C03642=1046.067,28.309,420.104,170.138,34.903,156.571
C03643=1046.061,28.059,420.121,170.136,34.901,156.571
C03644=1046.054,27.810,420.136,170.135,34.900,156.571
C03645=1046.047,27.560,420.153,170.133,34.899,156.571
C03646=1046.041,27.311,420.169,170.131,34.897,156.570
C03647=1046.035,27.062,420.185,170.130,34.895,156.570
C03648=1046.029,26.813,420.201,170.128,34.894,156.570
C03649=1046.022,26.564,420.217,170.126,34.893,156.570
C03650=1046.016,26.314,420.233,170.124,34.891,156.569
C03651=1046.010,26.064,420.250,170.123,34.889,156.569
C03652=1046.003,25.815,420.265,170.121,34.888,156.569
C03653=1045.997,25.566,420.281,170.119,34.887,156.569
C03654=1045.991,25.316,420.296,170.116,34.885,156.568
C03655=1045.985,25.067,420.313,170.115,34.883,156.568
C03656=1045.978,24.818,420.328,170.113,34.882,156.568
C03657=1045.971,24.568,420.345,170.111,34.881,156.568
C03658=1045.965,24.318,420.361,170.109,34.879,156.567
C03659=1045.959,24.069,420.377,170.108,34.878,156.567
C03660=1045.953,23.820,420.393,170.106,34.876,156.567
C03661=1045.946,23.570,420.408,170.104,34.875,156.567
C03662=1045.940,23.321,420.424,170.102,34.873,156.566
C03663=1045.934,23.072,420.440,170.101,34.872,156.566
C03664=1045.928,22.823,420.456,170.099,34.870,156.566
C03665=1045.921,22.572,420.473,170.097,34.869,156.566
C03666=1045.915,22.323,420.488,170.096,34.868,156.565
C03667=1045.909,22.073,420.504,170.094,34.866,156.565
C03668=1045.902,21.824,420.520,170.091,34.864,156.565
C03669=1045.896,21.575,420.536,170.089,34.863,156.565
C03670=1045.890,21.325,420.551,170.088,34.862,156.564
C03671=1045.884,21.076,420.567,170.086,34.860,156.564
C03672=1045.877,20.827,420.583,170.084,34.858,156.564
C03673=1045.871,20.578,420.599,170.082,34.857,156.564
C03674=1045.866,20.328,420.615,170.081,34.856,156.564
C03675=1045.859,20.079,420.630,170.079,34.854,156.563
C03676=1045.853,19.829,420.647,170.077,34.852,156.563
C03677=1045.846,19.579,420.662,170.075,34.851,156.563
C03678=1045.839,19.330,420.678,170.074,34.850,156.563
C03679=1045.833,19.081,420.694,170.072,34.848,156.562
C03680=1045.827,18.831,420.709,170.070,34.847,156.562
C03681=1045.821,18.582,420.725,170.068,34.846,156.562
C03682=1045.814,18.333,420.741,170.066,34.844,156.562
C03683=1045.808,18.083,420.756,170.064,34.842,156.561
C03684=1045.802,17.834,420.772,170.062,34.841,156.561
C03685=1045.795,17.585,420.788,170.060,34.840,156.561
C03686=1045.790,17.335,420.803,170.058,34.838,156.561
C03687=1045.783,17.086,420.819,170.057,34.837,156.561
C03688=1045.777,16.836,420.834,170.055,34.835,156.560
C03689=1045.771,16.586,420.850,170.053,34.834,156.560
C03690=1045.764,16.337,420.866,170.051,34.832,156.560
C03691=1045.758,16.087,420.881,170.050,34.831,156.560
C03692=1045.752,15.838,420.897,170.048,34.830,156.559
C03693=1045.745,15.589,420.912,170.046,34.828,156.559
C03694=1045.739,15.339,420.928,170.044,34.827,156.559
C03695=1045.733,15.090,420.943,170.043,34.825,156.559
C03696=1045.727,14.840,420.959,170.040,34.824,156.558
C03697=1045.721,14.591,420.974,170.038,34.823,156.558
C03698=1045.714,14.342,420.990,170.036,34.821,156.558
C03699=1045.708,14.092,421.005,170.035,34.820,156.558
C03700=1045.702,13.843,421.021,170.033,34.819,156.558
C03701=1045.695,13.593,421.036,170.031,34.817,156.557
C03702=1045.688,13.308,421.054,170.029,34.815,156.557
C03703=1045.680,13.023,421.071,170.027,34.814,156.557
C03704=1045.673,12.737,421.089,170.025,34.813,156.557
C03705=1045.666,12.453,421.106,170.023,34.811,156.556
C03706=1045.659,12.203,421.121,170.021,34.809,156.556
C03707=1045.653,11.954,421.138,170.019,34.808,156.556
C03708=1045.647,11.704,421.152,170.017,34.807,156.556
C03709=1045.640,11.455,421.167,170.015,34.805,156.555
C03710=1045.634,11.206,421.183,170.014,34.804,156.555
C03711=1045.627,10.956,421.198,170.011,34.803,156.555
C03712=1045.621,10.707,421.214,170.009,34.801,156.555
C03713=1045.614,10.457,421.229,170.007,34.800,156.555
C03714=1045.609,10.207,421.244,170.005,34.798,156.554
C03715=1045.602,9.958,421.260,170.004,34.797,156.554
C03716=1045.596,9.709,421.275,170.002,34.796,156.554
C03717=1045.589,9.459,421.290,170.000,34.795,156.554
C03718=1045.583,9.210,421.305,169.998,34.793,156.554
C03719=1045.576,8.960,421.320,169.996,34.792,156.553
C03720=1045.570,8.711,421.335,169.995,34.791,156.553
C03721=1045.563,8.462,421.351,169.993,34.789,156.553
C03722=1045.557,8.212,421.367,169.991,34.788,156.553
C03723=1045.551,7.962,421.381,169.989,34.786,156.552
C03724=1045.545,7.712,421.396,169.987,34.785,156.552
C03725=1045.538,7.463,421.412,169.986,34.783,156.552
C03726=1045.532,7.214,421.427,169.984,34.782,156.552
C03727=1045.526,6.965,421.442,169.981,34.780,156.552
C03728=1045.519,6.715,421.457,169.979,34.779,156.551
C03729=1045.513,6.466,421.472,169.977,34.778,156.551
C03730=1045.506,6.216,421.487,169.975,34.776,156.551
C03731=1045.501,5.966,421.503,169.974,34.775,156.551
C03732=1045.494,5.717,421.518,169.972,34.774,156.550
C03733=1045.488,5.468,421.533,169.970,34.772,156.550
C03734=1045.482,5.219,421.548,169.968,34.771,156.550
C03735=1045.476,4.969,421.563,169.966,34.770,156.550
C03736=1045.469,4.719,421.578,169.965,34.768,156.550
C03737=1045.463,4.470,421.593,169.963,34.767,156.549
C03738=1045.456,4.220,421.608,169.961,34.766,156.549
C03739=1045.450,3.971,421.623,169.959,34.764,156.549
C03740=1045.443,3.721,421.638,169.957,34.763,156.549
C03741=1045.437,3.472,421.653,169.955,34.762,156.549
C03742=1045.432,3.222,421.668,169.954,34.760,156.548
C03743=1045.425,2.973,421.683,169.952,34.759,156.548
C03744=1045.419,2.723,421.698,169.949,34.758,156.548
C03745=1045.413,2.473,421.713,169.947,34.756,156.548
C03746=1045.407,2.225,421.729,169.945,34.755,156.548
C03747=1045.400,1.975,421.743,169.943,34.754,156.547
C03748=1045.394,1.726,421.758,169.942,34.752,156.547
C03749=1045.387,1.476,421.773,169.940,34.751,156.547
C03750=1045.381,1.226,421.788,169.938,34.750,156.547
C03751=1045.375,0.977,421.803,169.936,34.748,156.546
C03752=1045.369,0.728,421.818,169.934,34.746,156.546
C03753=1045.363,0.478,421.833,169.932,34.745,156.546
C03754=1045.356,0.229,421.848,169.931,34.744,156.546
C03755=1045.350,-0.020,421.862,169.929,34.742,156.546
C03756=1045.344,-0.270,421.877,169.927,34.741,156.545
C03757=1045.338,-0.520,421.892,169.925,34.740,156.545
C03758=1045.332,-0.770,421.908,169.923,34.738,156.545
C03759=1045.326,-1.019,421.922,169.921,34.737,156.545
C03760=1045.320,-1.268,421.937,169.920,34.736,156.545
C03761=1045.313,-1.518,421.952,169.917,34.734,156.544
C03762=1045.307,-1.768,421.967,169.915,34.733,156.544
C03763=1045.301,-2.017,421.982,169.913,34.732,156.544
C03764=1045.295,-2.266,421.997,169.911,34.730,156.544
C03765=1045.288,-2.516,422.012,169.909,34.729,156.543
C03766=1045.281,-2.799,422.029,169.907,34.727,156.543
C03767=1045.274,-3.082,422.045,169.905,34.725,156.543
C03768=1045.267,-3.365,422.063,169.903,34.724,156.543
C03769=1045.260,-3.649,422.079,169.901,34.723,156.543
C03770=1045.254,-3.898,422.093,169.899,34.721,156.542
C03771=1045.247,-4.147,422.108,169.897,34.720,156.542
C03772=1045.241,-4.397,422.122,169.895,34.719,156.542
C03773=1045.235,-4.647,422.137,169.894,34.717,156.542
C03774=1045.228,-4.896,422.151,169.892,34.717,156.542
C03775=1045.222,-5.145,422.166,169.890,34.715,156.541
C03776=1045.216,-5.395,422.181,169.888,34.714,156.541
C03777=1045.209,-5.645,422.196,169.886,34.713,156.541
C03778=1045.203,-5.894,422.209,169.884,34.711,156.541
C03779=1045.197,-6.144,422.224,169.881,34.710,156.541
C03780=1045.190,-6.393,422.239,169.879,34.709,156.540
C03781=1045.184,-6.642,422.253,169.877,34.708,156.540
C03782=1045.177,-6.892,422.268,169.876,34.706,156.540
C03783=1045.171,-7.142,422.282,169.874,34.705,156.540
C03784=1045.165,-7.392,422.297,169.872,34.704,156.540
C03785=1045.158,-7.640,422.311,169.870,34.702,156.539
C03786=1045.152,-7.890,422.326,169.868,34.701,156.539
C03787=1045.146,-8.140,422.340,169.866,34.700,156.539
C03788=1045.139,-8.389,422.354,169.864,34.699,156.539
C03789=1045.133,-8.638,422.369,169.862,34.698,156.539
C03790=1045.127,-8.888,422.384,169.860,34.696,156.539
C03791=1045.121,-9.138,422.398,169.858,34.695,156.538
C03792=1045.114,-9.387,422.413,169.857,34.694,156.538
C03793=1045.108,-9.637,422.427,169.855,34.692,156.538
C03794=1045.102,-9.886,422.441,169.853,34.692,156.538
C03795=1045.095,-10.136,422.456,169.851,34.690,156.538
C03796=1045.089,-10.385,422.470,169.849,34.689,156.537
C03797=1045.083,-10.635,422.484,169.847,34.687,156.537
C03798=1045.076,-10.884,422.499,169.845,34.686,156.537
C03799=1045.070,-11.133,422.513,169.842,34.685,156.537
C03800=1045.064,-11.383,422.528,169.840,34.684,156.537
C03801=1045.058,-11.633,422.543,169.838,34.683,156.536
C03802=1045.052,-11.882,422.556,169.837,34.681,156.536
C03803=1045.045,-12.132,422.571,169.835,34.680,156.536
C03804=1045.039,-12.381,422.585,169.833,34.679,156.536
C03805=1045.033,-12.631,422.599,169.831,34.677,156.536
C03806=1045.027,-12.880,422.614,169.829,34.677,156.536
C03807=1045.021,-13.130,422.628,169.827,34.675,156.535
C03808=1045.014,-13.379,422.642,169.825,34.674,156.535
C03809=1045.008,-13.628,422.657,169.823,34.672,156.535
C03810=1045.002,-13.879,422.671,169.821,34.671,156.535
C03811=1044.995,-14.127,422.685,169.819,34.670,156.535
C03812=1044.989,-14.378,422.699,169.817,34.669,156.534
C03813=1044.983,-14.627,422.714,169.816,34.668,156.534
C03814=1044.977,-14.877,422.727,169.814,34.666,156.534
C03815=1044.971,-15.125,422.742,169.812,34.665,156.534
C03816=1044.964,-15.375,422.756,169.810,34.664,156.534
C03817=1044.958,-15.625,422.771,169.808,34.663,156.534
C03818=1044.951,-15.874,422.784,169.806,34.662,156.533
C03819=1044.945,-16.124,422.799,169.804,34.660,156.533
C03820=1044.939,-16.373,422.812,169.801,34.659,156.533
C03821=1044.933,-16.624,422.826,169.799,34.658,156.533
C03822=1044.926,-16.872,422.840,169.797,34.657,156.533
C03823=1044.919,-17.122,422.854,169.795,34.656,156.533
C03824=1044.913,-17.372,422.869,169.793,34.655,156.532
C03825=1044.907,-17.621,422.882,169.791,34.653,156.532
C03826=1044.900,-17.871,422.897,169.789,34.653,156.532
C03827=1044.894,-18.120,422.910,169.787,34.651,156.532
C03828=1044.888,-18.370,422.925,169.785,34.650,156.532
C03829=1044.882,-18.619,422.939,169.783,34.648,156.531
C03830=1044.874,-18.901,422.954,169.781,34.648,156.531
C03831=1044.867,-19.183,422.970,169.779,34.646,156.531
C03832=1044.860,-19.464,422.986,169.777,34.645,156.531
C03833=1044.853,-19.745,423.002,169.775,34.644,156.531
C03834=1044.847,-19.996,423.016,169.773,34.642,156.530
C03835=1044.841,-20.245,423.029,169.771,34.642,156.530
C03836=1044.834,-20.495,423.043,169.769,34.640,156.530
C03837=1044.828,-20.744,423.057,169.767,34.639,156.530
C03838=1044.821,-20.994,423.071,169.765,34.638,156.530
C03839=1044.816,-21.243,423.085,169.763,34.637,156.530
C03840=1044.809,-21.493,423.099,169.761,34.635,156.529
C03841=1044.803,-21.742,423.112,169.759,34.635,156.529
C03842=1044.796,-21.992,423.127,169.757,34.633,156.529
C03843=1044.790,-22.242,423.140,169.755,34.632,156.529
C03844=1044.784,-22.491,423.154,169.752,34.631,156.529
C03845=1044.778,-22.741,423.168,169.750,34.630,156.529
C03846=1044.771,-22.990,423.181,169.748,34.628,156.528
C03847=1044.765,-23.240,423.196,169.746,34.628,156.528
C03848=1044.759,-23.489,423.210,169.744,34.626,156.528
C03849=1044.752,-23.739,423.223,169.742,34.625,156.528
C03850=1044.747,-23.988,423.237,169.740,34.624,156.528
C03851=1044.740,-24.238,423.250,169.738,34.623,156.528
C03852=1044.734,-24.488,423.265,169.736,34.621,156.527
C03853=1044.728,-24.736,423.279,169.734,34.621,156.527
C03854=1044.721,-24.986,423.292,169.732,34.619,156.527
C03855=1044.715,-25.236,423.306,169.730,34.618,156.527
C03856=1044.709,-25.485,423.319,169.728,34.617,156.527
C03857=1044.702,-25.735,423.333,169.726,34.616,156.527
C03858=1044.697,-25.985,423.347,169.724,34.615,156.527
C03859=1044.691,-26.234,423.360,169.722,34.614,156.526
C03860=1044.684,-26.483,423.374,169.720,34.612,156.526
C03861=1044.678,-26.733,423.388,169.718,34.611,156.526
C03862=1044.672,-26.982,423.402,169.716,34.610,156.526
C03863=1044.665,-27.232,423.415,169.714,34.609,156.526
C03864=1044.659,-27.481,423.428,169.712,34.608,156.526
C03865=1044.653,-27.732,423.443,169.710,34.607,156.525
C03866=1044.647,-27.981,423.456,169.708,34.606,156.525
C03867=1044.640,-28.230,423.469,169.706,34.605,156.525
C03868=1044.634,-28.480,423.483,169.704,34.604,156.525
C03869=1044.627,-28.729,423.496,169.702,34.603,156.525
C03870=1044.621,-28.979,423.510,169.700,34.602,156.525
C03871=1044.614,-29.229,423.523,169.697,34.601,156.525
C03872=1044.608,-29.478,423.536,169.695,34.600,156.524
C03873=1044.601,-29.728,423.550,169.693,34.598,156.524
C03874=1044.596,-29.978,423.564,169.691,34.598,156.524
C03875=1044.590,-30.227,423.577,169.689,34.596,156.524
C03876=1044.583,-30.477,423.591,169.687,34.596,156.524
C03877=1044.577,-30.726,423.604,169.685,34.594,156.524
C03878=1044.570,-30.975,423.617,169.683,34.594,156.524
C03879=1044.564,-31.225,423.631,169.681,34.593,156.523
C03880=1044.557,-31.475,423.644,169.679,34.591,156.523
C03881=1044.551,-31.724,423.657,169.677,34.591,156.523
C03882=1044.545,-31.974,423.670,169.675,34.589,156.523
C03883=1044.539,-32.224,423.684,169.673,34.589,156.523
C03884=1044.533,-32.473,423.698,169.671,34.587,156.523
C03885=1044.527,-32.722,423.711,169.669,34.587,156.523
C03886=1044.520,-32.972,423.724,169.667,34.585,156.522
C03887=1044.514,-33.222,423.738,169.665,34.584,156.522
C03888=1044.507,-33.471,423.751,169.663,34.583,156.522
C03889=1044.501,-33.721,423.765,169.660,34.582,156.522
C03890=1044.495,-33.971,423.777,169.658,34.581,156.522
C03891=1044.488,-34.220,423.790,169.656,34.580,156.522
C03892=1044.482,-34.469,423.804,169.654,34.579,156.522
C03893=1044.475,-34.719,423.817,169.652,34.578,156.521
C03894=1044.468,-35.047,423.834,169.650,34.577,156.521
C03895=1044.460,-35.375,423.852,169.647,34.575,156.521
C03896=1044.451,-35.704,423.869,169.644,34.574,156.521
C03897=1044.443,-36.032,423.887,169.642,34.572,156.521
C03898=1044.437,-36.258,423.898,169.640,34.572,156.521
C03899=1044.432,-36.484,423.911,169.638,34.571,156.520
C03900=1044.426,-36.710,423.923,169.636,34.570,156.520
C03901=1044.421,-36.935,423.934,169.634,34.569,156.520
C03902=1044.415,-37.161,423.947,169.632,34.568,156.520
C03903=1044.410,-37.387,423.959,169.630,34.567,156.520
C03904=1044.404,-37.613,423.971,169.628,34.566,156.520
C03905=1044.398,-37.839,423.982,169.626,34.565,156.520
C03906=1044.392,-38.089,423.996,169.624,34.564,156.520
C03907=1044.385,-38.338,424.009,169.622,34.563,156.519
C03908=1044.379,-38.588,424.021,169.619,34.562,156.519
C03909=1044.373,-38.837,424.035,169.617,34.561,156.519
C03910=1044.367,-39.087,424.048,169.615,34.560,156.519
C03911=1044.361,-39.337,424.061,169.613,34.560,156.519
C03912=1044.354,-39.586,424.074,169.611,34.558,156.519
C03913=1044.348,-39.836,424.087,169.609,34.557,156.519
C03914=1044.341,-40.085,424.099,169.607,34.557,156.519
C03915=1044.335,-40.335,424.113,169.605,34.556,156.518
C03916=1044.329,-40.584,424.125,169.603,34.555,156.518
C03917=1044.322,-40.834,424.139,169.601,34.554,156.518
C03918=1044.317,-41.084,424.151,169.599,34.553,156.518
C03919=1044.310,-41.333,424.164,169.596,34.552,156.518
C03920=1044.303,-41.583,424.177,169.594,34.551,156.518
C03921=1044.298,-41.832,424.190,169.592,34.550,156.518
C03922=1044.291,-42.082,424.203,169.590,34.549,156.518
C03923=1044.285,-42.332,424.216,169.588,34.548,156.517
C03924=1044.279,-42.582,424.229,169.586,34.547,156.517
C03925=1044.272,-42.831,424.241,169.584,34.547,156.517
C03926=1044.266,-43.080,424.255,169.582,34.546,156.517
C03927=1044.260,-43.330,424.267,169.580,34.545,156.517
C03928=1044.254,-43.579,424.280,169.578,34.544,156.517
C03929=1044.247,-43.829,424.292,169.575,34.543,156.517
C03930=1044.241,-44.078,424.306,169.573,34.542,156.517
C03931=1044.234,-44.329,424.319,169.571,34.541,156.517
C03932=1044.228,-44.578,424.332,169.569,34.540,156.516
C03933=1044.222,-44.828,424.344,169.567,34.539,156.516
C03934=1044.215,-45.077,424.357,169.565,34.539,156.516
C03935=1044.209,-45.327,424.370,169.563,34.537,156.516
C03936=1044.203,-45.577,424.382,169.561,34.537,156.516
C03937=1044.197,-45.826,424.395,169.559,34.536,156.516
C03938=1044.190,-46.076,424.407,169.556,34.535,156.516
C03939=1044.184,-46.325,424.421,169.554,34.534,156.516
C03940=1044.178,-46.575,424.433,169.552,34.533,156.516
C03941=1044.172,-46.825,424.446,169.550,34.532,156.515
C03942=1044.166,-47.074,424.459,169.548,34.531,156.515
C03943=1044.160,-47.323,424.471,169.546,34.531,156.515
C03944=1044.153,-47.573,424.484,169.544,34.529,156.515
C03945=1044.147,-47.823,424.497,169.542,34.529,156.515
C03946=1044.142,-48.073,424.509,169.540,34.528,156.515
C03947=1044.135,-48.321,424.522,169.537,34.527,156.515
C03948=1044.129,-48.571,424.535,169.534,34.526,156.515
C03949=1044.123,-48.821,424.547,169.532,34.525,156.515
C03950=1044.117,-49.070,424.560,169.530,34.524,156.514
C03951=1044.110,-49.320,424.572,169.528,34.523,156.514
C03952=1044.104,-49.570,424.585,169.526,34.523,156.514
C03953=1044.098,-49.819,424.598,169.524,34.521,156.514
C03954=1044.092,-50.069,424.611,169.522,34.521,156.514
C03955=1044.085,-50.319,424.623,169.519,34.520,156.514
C03956=1044.079,-50.569,424.635,169.517,34.519,156.514
C03957=1044.073,-50.818,424.647,169.515,34.518,156.514
C03958=1044.065,-51.100,424.662,169.513,34.518,156.514
C03959=1044.058,-51.381,424.676,169.510,34.517,156.514
C03960=1044.052,-51.662,424.689,169.508,34.516,156.513
C03961=1044.043,-51.943,424.703,169.505,34.515,156.513
C03962=1044.038,-52.193,424.716,169.503,34.514,156.513
C03963=1044.031,-52.443,424.728,169.501,34.514,156.513
C03964=1044.025,-52.692,424.741,169.499,34.513,156.513
C03965=1044.018,-52.942,424.753,169.497,34.512,156.513
C03966=1044.011,-53.191,424.765,169.494,34.511,156.513
C03967=1044.005,-53.441,424.778,169.492,34.511,156.513
C03968=1043.999,-53.691,424.790,169.490,34.510,156.513
C03969=1043.993,-53.941,424.802,169.488,34.509,156.513
C03970=1043.986,-54.190,424.814,169.486,34.508,156.513
C03971=1043.980,-54.440,424.826,169.483,34.508,156.513
C03972=1043.974,-54.690,424.839,169.481,34.507,156.512
C03973=1043.967,-54.939,424.851,169.479,34.506,156.512
C03974=1043.960,-55.188,424.863,169.477,34.505,156.512
C03975=1043.954,-55.438,424.876,169.475,34.505,156.512
C03976=1043.948,-55.688,424.888,169.473,34.504,156.512
C03977=1043.942,-55.937,424.900,169.470,34.503,156.512
C03978=1043.935,-56.187,424.912,169.468,34.502,156.512
C03979=1043.928,-56.437,424.924,169.466,34.502,156.512
C03980=1043.923,-56.686,424.936,169.464,34.501,156.512
C03981=1043.916,-56.935,424.948,169.462,34.501,156.512
C03982=1043.910,-57.185,424.960,169.459,34.500,156.512
C03983=1043.904,-57.435,424.973,169.457,34.499,156.512
C03984=1043.897,-57.684,424.985,169.455,34.499,156.512
C03985=1043.891,-57.934,424.997,169.453,34.498,156.511
C03986=1043.885,-58.184,425.009,169.451,34.497,156.511
C03987=1043.878,-58.433,425.021,169.448,34.496,156.511
C03988=1043.872,-58.683,425.034,169.446,34.495,156.511
C03989=1043.866,-58.933,425.045,169.444,34.495,156.511
C03990=1043.860,-59.182,425.057,169.442,34.494,156.511
C03991=1043.854,-59.432,425.069,169.440,34.493,156.511
C03992=1043.847,-59.682,425.081,169.437,34.493,156.511
C03993=1043.840,-59.931,425.093,169.435,34.492,156.511
C03994=1043.835,-60.181,425.106,169.433,34.492,156.511
C03995=1043.828,-60.431,425.118,169.431,34.491,156.511
C03996=1043.822,-60.680,425.129,169.429,34.490,156.511
C03997=1043.816,-60.930,425.142,169.426,34.489,156.511
C03998=1043.809,-61.179,425.154,169.424,34.489,156.510
C03999=1043.803,-61.429,425.165,169.422,34.488,156.510
C04000=1043.797,-61.679,425.178,169.420,34.487,156.510
C04001=1043.791,-61.928,425.189,169.418,34.487,156.510
C04002=1043.784,-62.178,425.201,169.415,34.486,156.510
C04003=1043.778,-62.428,425.214,169.413,34.485,156.510
C04004=1043.772,-62.677,425.226,169.411,34.485,156.510
C04005=1043.765,-62.927,425.237,169.409,34.484,156.510
C04006=1043.760,-63.177,425.249,169.406,34.483,156.510
C04007=1043.754,-63.426,425.261,169.404,34.482,156.510
C04008=1043.747,-63.676,425.273,169.402,34.482,156.510
C04009=1043.740,-63.925,425.285,169.400,34.482,156.510
C04010=1043.735,-64.175,425.296,169.398,34.481,156.510
C04011=1043.729,-64.425,425.308,169.395,34.480,156.510
C04012=1043.722,-64.674,425.320,169.393,34.479,156.509
C04013=1043.716,-64.924,425.333,169.391,34.479,156.509
C04014=1043.710,-65.174,425.344,169.389,34.478,156.509
C04015=1043.704,-65.423,425.356,169.386,34.478,156.509
C04016=1043.698,-65.673,425.368,169.384,34.477,156.509
C04017=1043.691,-65.923,425.380,169.382,34.476,156.509
C04018=1043.685,-66.172,425.391,169.380,34.475,156.509
C04019=1043.679,-66.422,425.403,169.378,34.475,156.509
C04020=1043.673,-66.672,425.416,169.375,34.474,156.509
C04021=1043.667,-66.921,425.426,169.373,34.474,156.509
C04022=1043.659,-67.204,425.441,169.371,34.473,156.509
C04023=1043.653,-67.486,425.454,169.368,34.472,156.509
C04024=1043.646,-67.769,425.467,169.366,34.471,156.509
C04025=1043.639,-68.051,425.480,169.363,34.471,156.509
C04026=1043.633,-68.301,425.492,169.361,34.470,156.509
C04027=1043.627,-68.550,425.503,169.359,34.469,156.508
C04028=1043.621,-68.800,425.516,169.356,34.469,156.509
C04029=1043.614,-69.050,425.527,169.354,34.468,156.508
C04030=1043.608,-69.299,425.539,169.352,34.467,156.508
C04031=1043.603,-69.550,425.550,169.350,34.467,156.508
C04032=1043.596,-69.799,425.562,169.347,34.467,156.508
C04033=1043.590,-70.049,425.573,169.345,34.466,156.508
C04034=1043.584,-70.298,425.585,169.343,34.465,156.508
C04035=1043.578,-70.548,425.597,169.341,34.464,156.508
C04036=1043.572,-70.798,425.609,169.338,34.463,156.508
C04037=1043.565,-71.047,425.621,169.336,34.463,156.508
C04038=1043.560,-71.297,425.631,169.334,34.463,156.508
C04039=1043.553,-71.546,425.643,169.332,34.462,156.508
C04040=1043.548,-71.796,425.655,169.329,34.461,156.508
C04041=1043.541,-72.046,425.667,169.327,34.461,156.508
C04042=1043.535,-72.296,425.678,169.325,34.460,156.508
C04043=1043.529,-72.545,425.690,169.323,34.459,156.508
C04044=1043.523,-72.795,425.701,169.320,34.459,156.508
C04045=1043.517,-73.044,425.713,169.318,34.459,156.508
C04046=1043.511,-73.294,425.724,169.316,34.458,156.507
C04047=1043.505,-73.543,425.736,169.314,34.457,156.507
C04048=1043.499,-73.794,425.748,169.311,34.456,156.507
C04049=1043.493,-74.044,425.759,169.309,34.456,156.507
C04050=1043.487,-74.293,425.771,169.307,34.455,156.507
C04051=1043.481,-74.543,425.782,169.305,34.455,156.507
C04052=1043.474,-74.792,425.793,169.302,34.455,156.507
C04053=1043.468,-75.042,425.805,169.300,34.454,156.507
C04054=1043.462,-75.292,425.816,169.298,34.454,156.507
C04055=1043.456,-75.541,425.827,169.295,34.453,156.507
C04056=1043.449,-75.791,425.839,169.293,34.453,156.507
C04057=1043.444,-76.041,425.850,169.291,34.452,156.507
C04058=1043.436,-76.290,425.861,169.289,34.452,156.507
C04059=1043.431,-76.540,425.872,169.286,34.451,156.507
C04060=1043.424,-76.790,425.883,169.284,34.451,156.507
C04061=1043.418,-77.039,425.895,169.282,34.450,156.507
C04062=1043.412,-77.289,425.906,169.279,34.450,156.507
C04063=1043.406,-77.538,425.917,169.277,34.449,156.507
C04064=1043.399,-77.788,425.929,169.275,34.449,156.507
C04065=1043.394,-78.037,425.940,169.272,34.448,156.507
C04066=1043.387,-78.288,425.951,169.270,34.448,156.507
C04067=1043.382,-78.537,425.962,169.268,34.448,156.507
C04068=1043.375,-78.787,425.974,169.266,34.447,156.507
C04069=1043.369,-79.036,425.985,169.263,34.447,156.507
C04070=1043.363,-79.286,425.996,169.261,34.446,156.507
C04071=1043.357,-79.536,426.007,169.259,34.446,156.507
C04072=1043.351,-79.786,426.018,169.256,34.445,156.507
C04073=1043.345,-80.035,426.030,169.254,34.445,156.507
C04074=1043.338,-80.285,426.040,169.252,34.445,156.507
C04075=1043.331,-80.535,426.051,169.249,34.444,156.507
C04076=1043.326,-80.784,426.062,169.247,34.444,156.507
C04077=1043.319,-81.034,426.073,169.245,34.444,156.507
C04078=1043.313,-81.284,426.084,169.242,34.443,156.506
C04079=1043.306,-81.534,426.095,169.240,34.443,156.507
C04080=1043.301,-81.783,426.106,169.238,34.443,156.507
C04081=1043.293,-82.033,426.117,169.235,34.442,156.506
C04082=1043.288,-82.282,426.128,169.233,34.442,156.507
C04083=1043.282,-82.532,426.139,169.231,34.442,156.507
C04084=1043.275,-82.782,426.150,169.228,34.441,156.506
C04085=1043.269,-83.031,426.161,169.226,34.441,156.506
C04086=1043.262,-83.316,426.173,169.223,34.441,156.507
C04087=1043.255,-83.600,426.186,169.221,34.440,156.506
C04088=1043.247,-83.886,426.198,169.218,34.440,156.506
C04089=1043.240,-84.171,426.210,169.215,34.439,156.507
C04090=1043.234,-84.421,426.221,169.213,34.439,156.506
C04091=1043.229,-84.670,426.232,169.211,34.439,156.506
C04092=1043.221,-84.920,426.243,169.208,34.438,156.506
C04093=1043.216,-85.169,426.253,169.206,34.438,156.507
C04094=1043.209,-85.420,426.265,169.204,34.438,156.506
C04095=1043.203,-85.669,426.275,169.201,34.437,156.506
C04096=1043.197,-85.918,426.286,169.199,34.437,156.506
C04097=1043.191,-86.169,426.297,169.197,34.437,156.507
C04098=1043.184,-86.418,426.307,169.194,34.436,156.506
C04099=1043.178,-86.668,426.319,169.192,34.436,156.506
C04100=1043.172,-86.917,426.330,169.190,34.436,156.506
C04101=1043.166,-87.167,426.340,169.187,34.436,156.507
C04102=1043.159,-87.417,426.351,169.185,34.435,156.506
C04103=1043.153,-87.666,426.361,169.182,34.435,156.506
C04104=1043.147,-87.915,426.372,169.180,34.435,156.507
C04105=1043.141,-88.166,426.383,169.178,34.435,156.507
C04106=1043.134,-88.415,426.394,169.175,34.434,156.506
C04107=1043.129,-88.665,426.404,169.173,34.434,156.506
C04108=1043.123,-88.915,426.415,169.171,34.434,156.507
C04109=1043.116,-89.164,426.425,169.168,34.434,156.507
C04110=1043.110,-89.414,426.436,169.166,34.434,156.507
C04111=1043.104,-89.664,426.448,169.164,34.433,156.506
C04112=1043.098,-89.913,426.458,169.161,34.433,156.507
C04113=1043.092,-90.163,426.469,169.159,34.433,156.507
C04114=1043.086,-90.413,426.479,169.157,34.432,156.507
C04115=1043.079,-90.663,426.490,169.154,34.432,156.507
C04116=1043.074,-90.912,426.500,169.152,34.432,156.507
C04117=1043.067,-91.161,426.511,169.150,34.431,156.507
C04118=1043.061,-91.411,426.522,169.147,34.431,156.507
C04119=1043.055,-91.662,426.532,169.145,34.431,156.507
C04120=1043.049,-91.911,426.542,169.142,34.431,156.507
C04121=1043.043,-92.161,426.554,169.140,34.430,156.507
C04122=1043.036,-92.410,426.564,169.138,34.430,156.507
C04123=1043.031,-92.660,426.574,169.136,34.430,156.507
C04124=1043.025,-92.910,426.585,169.134,34.430,156.507
C04125=1043.018,-93.160,426.596,169.132,34.430,156.507
C04126=1043.012,-93.409,426.606,169.129,34.430,156.507
C04127=1043.006,-93.659,426.616,169.127,34.429,156.507
C04128=1043.000,-93.908,426.627,169.124,34.429,156.507
C04129=1042.994,-94.158,426.638,169.122,34.429,156.507
C04130=1042.988,-94.408,426.648,169.120,34.428,156.507
C04131=1042.982,-94.658,426.659,169.117,34.428,156.507
C04132=1042.975,-94.907,426.669,169.115,34.428,156.507
C04133=1042.970,-95.157,426.679,169.113,34.428,156.507
C04134=1042.964,-95.407,426.690,169.110,34.427,156.507
C04135=1042.957,-95.657,426.701,169.108,34.427,156.507
C04136=1042.952,-95.907,426.711,169.106,34.427,156.507
C04137=1042.945,-96.156,426.721,169.103,34.427,156.507
C04138=1042.940,-96.405,426.732,169.101,34.427,156.507
C04139=1042.933,-96.655,426.741,169.098,34.427,156.507
C04140=1042.928,-96.905,426.752,169.096,34.426,156.507
C04141=1042.922,-97.155,426.763,169.094,34.426,156.507
C04142=1042.915,-97.405,426.773,169.091,34.426,156.507
C04143=1042.909,-97.654,426.784,169.089,34.426,156.507
C04144=1042.903,-97.904,426.794,169.086,34.426,156.507
C04145=1042.897,-98.153,426.804,169.084,34.426,156.507
C04146=1042.891,-98.403,426.814,169.082,34.426,156.507
C04147=1042.884,-98.653,426.825,169.079,34.425,156.507
C04148=1042.878,-98.903,426.834,169.077,34.425,156.507
C04149=1042.872,-99.152,426.845,169.074,34.425,156.507
C04150=1042.865,-99.440,426.856,169.072,34.425,156.507
C04151=1042.857,-99.726,426.868,169.069,34.425,156.507
C04152=1042.851,-100.013,426.880,169.066,34.425,156.507
C04153=1042.844,-100.301,426.891,169.063,34.425,156.507
C04154=1042.838,-100.550,426.901,169.061,34.425,156.508
C04155=1042.832,-100.801,426.912,169.059,34.425,156.508
C04156=1042.825,-101.050,426.922,169.056,34.425,156.508
C04157=1042.819,-101.300,426.932,169.054,34.425,156.508
C04158=1042.813,-101.550,426.942,169.051,34.425,156.508
C04159=1042.807,-101.799,426.952,169.049,34.424,156.508
C04160=1042.801,-102.049,426.962,169.046,34.424,156.508
C04161=1042.794,-102.298,426.972,169.044,34.424,156.508
C04162=1042.789,-102.548,426.982,169.042,34.425,156.508
C04163=1042.783,-102.798,426.992,169.039,34.425,156.508
C04164=1042.776,-103.047,427.002,169.037,34.424,156.508
C04165=1042.770,-103.298,427.012,169.034,34.424,156.508
C04166=1042.764,-103.547,427.023,169.032,34.424,156.508
C04167=1042.758,-103.797,427.032,169.030,34.424,156.508
C04168=1042.752,-104.047,427.043,169.027,34.424,156.508
C04169=1042.746,-104.296,427.053,169.026,34.424,156.508
C04170=1042.739,-104.546,427.062,169.023,34.424,156.508
C04171=1042.733,-104.796,427.072,169.021,34.424,156.508
C04172=1042.728,-105.046,427.082,169.018,34.424,156.508
C04173=1042.721,-105.295,427.092,169.016,34.424,156.508
C04174=1042.715,-105.545,427.102,169.014,34.424,156.508
C04175=1042.709,-105.794,427.111,169.011,34.424,156.509
C04176=1042.703,-106.044,427.122,169.009,34.424,156.509
C04177=1042.697,-106.294,427.132,169.006,34.424,156.509
C04178=1042.691,-106.544,427.142,169.004,34.424,156.509
C04179=1042.685,-106.793,427.151,169.001,34.424,156.509
C04180=1042.679,-107.043,427.161,168.999,34.424,156.509
C04181=1042.673,-107.293,427.172,168.997,34.424,156.509
C04182=1042.667,-107.542,427.181,168.994,34.425,156.509
C04183=1042.661,-107.792,427.191,168.992,34.424,156.509
C04184=1042.654,-108.042,427.200,168.989,34.424,156.509
C04185=1042.648,-108.292,427.210,168.987,34.425,156.509
C04186=1042.642,-108.541,427.220,168.984,34.425,156.509
C04187=1042.636,-108.791,427.230,168.982,34.425,156.509
C04188=1042.629,-109.041,427.239,168.979,34.425,156.509
C04189=1042.624,-109.291,427.249,168.977,34.425,156.509
C04190=1042.618,-109.540,427.259,168.975,34.425,156.509
C04191=1042.612,-109.790,427.269,168.972,34.425,156.510
C04192=1042.605,-110.040,427.278,168.970,34.425,156.510
C04193=1042.599,-110.290,427.288,168.967,34.425,156.510
C04194=1042.593,-110.540,427.297,168.965,34.426,156.510
C04195=1042.587,-110.789,427.307,168.962,34.425,156.510
C04196=1042.580,-111.039,427.317,168.960,34.426,156.510
C04197=1042.574,-111.288,427.327,168.957,34.426,156.510
C04198=1042.568,-111.538,427.336,168.955,34.426,156.510
C04199=1042.562,-111.788,427.346,168.952,34.426,156.510
C04200=1042.556,-112.037,427.355,168.950,34.426,156.510
C04201=1042.550,-112.287,427.365,168.949,34.427,156.510
C04202=1042.544,-112.537,427.374,168.946,34.426,156.510
C04203=1042.539,-112.787,427.384,168.944,34.426,156.510
C04204=1042.532,-113.037,427.394,168.941,34.427,156.511
C04205=1042.526,-113.286,427.403,168.939,34.427,156.511
C04206=1042.520,-113.536,427.413,168.936,34.427,156.511
C04207=1042.514,-113.786,427.423,168.934,34.427,156.511
C04208=1042.508,-114.036,427.432,168.931,34.427,156.511
C04209=1042.502,-114.286,427.442,168.929,34.427,156.511
C04210=1042.496,-114.535,427.451,168.926,34.427,156.511
C04211=1042.490,-114.785,427.460,168.924,34.428,156.511
C04212=1042.484,-115.034,427.470,168.921,34.428,156.511
C04213=1042.477,-115.284,427.480,168.919,34.428,156.511
C04214=1042.470,-115.570,427.490,168.916,34.429,156.511
C04215=1042.463,-115.857,427.501,168.913,34.428,156.511
C04216=1042.456,-116.142,427.511,168.910,34.429,156.512
C04217=1042.449,-116.429,427.522,168.908,34.429,156.512
C04218=1042.443,-116.678,427.532,168.905,34.429,156.512
C04219=1042.437,-116.928,427.541,168.903,34.430,156.512
C04220=1042.431,-117.179,427.550,168.900,34.430,156.512
C04221=1042.426,-117.428,427.559,168.898,34.430,156.512
C04222=1042.420,-117.677,427.569,168.895,34.430,156.512
C04223=1042.413,-117.927,427.579,168.893,34.431,156.512
C04224=1042.406,-118.177,427.587,168.890,34.430,156.512
C04225=1042.400,-118.427,427.597,168.888,34.431,156.512
C04226=1042.394,-118.677,427.606,168.885,34.431,156.513
C04227=1042.389,-118.926,427.615,168.883,34.431,156.513
C04228=1042.383,-119.176,427.625,168.881,34.432,156.513
C04229=1042.376,-119.426,427.634,168.879,34.432,156.513
C04230=1042.371,-119.676,427.643,168.876,34.432,156.513
C04231=1042.364,-119.926,427.652,168.874,34.433,156.513
C04232=1042.358,-120.175,427.661,168.871,34.433,156.513
C04233=1042.352,-120.424,427.671,168.869,34.433,156.513
C04234=1042.346,-120.675,427.680,168.866,34.434,156.513
C04235=1042.340,-120.925,427.689,168.864,34.433,156.513
C04236=1042.334,-121.174,427.698,168.861,34.434,156.514
C04237=1042.328,-121.424,427.708,168.859,34.434,156.514
C04238=1042.322,-121.674,427.716,168.857,34.434,156.514
C04239=1042.315,-121.923,427.726,168.854,34.435,156.514
C04240=1042.310,-122.173,427.735,168.852,34.435,156.514
C04241=1042.304,-122.423,427.744,168.849,34.435,156.514
C04242=1042.298,-122.673,427.753,168.847,34.436,156.514
C04243=1042.291,-122.922,427.762,168.844,34.436,156.514
C04244=1042.286,-123.172,427.771,168.842,34.437,156.514
C04245=1042.279,-123.422,427.780,168.839,34.437,156.515
C04246=1042.273,-123.672,427.790,168.837,34.437,156.515
C04247=1042.268,-123.921,427.799,168.834,34.438,156.515
C04248=1042.261,-124.171,427.808,168.832,34.438,156.515
C04249=1042.255,-124.421,427.816,168.829,34.438,156.515
C04250=1042.249,-124.671,427.826,168.827,34.439,156.515
C04251=1042.243,-124.920,427.835,168.824,34.439,156.515
C04252=1042.237,-125.170,427.843,168.823,34.440,156.515
C04253=1042.231,-125.420,427.853,168.820,34.439,156.515
C04254=1042.225,-125.670,427.861,168.818,34.440,156.516
C04255=1042.219,-125.919,427.870,168.815,34.440,156.516
C04256=1042.213,-126.170,427.879,168.813,34.441,156.516
C04257=1042.207,-126.419,427.888,168.810,34.441,156.516
C04258=1042.200,-126.669,427.897,168.807,34.442,156.516
C04259=1042.194,-126.919,427.906,168.805,34.442,156.516
C04260=1042.189,-127.168,427.915,168.802,34.442,156.516
C04261=1042.182,-127.418,427.924,168.800,34.443,156.516
C04262=1042.176,-127.668,427.933,168.797,34.443,156.517
C04263=1042.171,-127.917,427.942,168.795,34.444,156.517
C04264=1042.166,-128.167,427.952,168.793,34.444,156.517
C04265=1042.162,-128.416,427.962,168.790,34.443,156.517
C04266=1042.158,-128.667,427.973,168.788,34.442,156.516
C04267=1042.156,-128.917,427.985,168.786,34.440,156.516
C04268=1042.154,-129.166,427.996,168.785,34.438,156.516
C04269=1042.153,-129.417,428.008,168.783,34.436,156.516
C04270=1042.153,-129.667,428.022,168.781,34.433,156.515
C04271=1042.155,-129.917,428.035,168.780,34.429,156.515
C04272=1042.157,-130.167,428.050,168.778,34.425,156.514
C04273=1042.159,-130.417,428.065,168.777,34.422,156.513
C04274=1042.163,-130.667,428.080,168.776,34.417,156.513
C04275=1042.167,-130.918,428.097,168.775,34.412,156.512
C04276=1042.172,-131.168,428.114,168.774,34.406,156.511
C04277=1042.179,-131.418,428.132,168.772,34.400,156.510
C04278=1041.829,-131.442,427.879,168.725,34.589,156.543
C04279=1041.823,-131.192,427.862,168.727,34.596,156.544
C04280=1041.817,-130.942,427.844,168.728,34.601,156.545
C04281=1041.813,-130.691,427.828,168.729,34.606,156.546
C04282=1041.810,-130.441,427.812,168.730,34.612,156.547
C04283=1041.807,-130.191,427.797,168.731,34.616,156.547
C04284=1041.805,-129.941,427.783,168.733,34.620,156.548
C04285=1041.804,-129.691,427.769,168.734,34.623,156.548
C04286=1041.804,-129.441,427.756,168.736,34.626,156.549
C04287=1041.804,-129.191,427.743,168.738,34.628,156.549
C04288=1041.806,-128.940,427.731,168.739,34.630,156.550
C04289=1041.808,-128.691,427.719,168.741,34.632,156.550
C04290=1041.812,-128.441,427.708,168.743,34.633,156.550
C04291=1041.816,-128.191,427.698,168.746,34.633,156.550
C04292=1041.821,-127.942,427.688,168.748,34.633,156.550
C04293=1041.826,-127.692,427.680,168.750,34.633,156.550
C04294=1041.832,-127.442,427.670,168.753,34.633,156.550
C04295=1041.839,-127.192,427.662,168.756,34.632,156.550
C04296=1041.844,-126.943,427.653,168.758,34.632,156.549
C04297=1041.850,-126.693,427.644,168.761,34.631,156.549
C04298=1041.857,-126.443,427.635,168.763,34.631,156.549
C04299=1041.862,-126.193,427.626,168.766,34.630,156.549
C04300=1041.868,-125.944,427.617,168.768,34.630,156.549
C04301=1041.875,-125.693,427.608,168.771,34.630,156.549
C04302=1041.881,-125.444,427.599,168.773,34.629,156.549
C04303=1041.887,-125.194,427.590,168.776,34.629,156.549
C04304=1041.893,-124.944,427.581,168.778,34.628,156.548
C04305=1041.899,-124.695,427.572,168.781,34.628,156.548
C04306=1041.905,-124.445,427.563,168.782,34.627,156.548
C04307=1041.911,-124.195,427.554,168.785,34.627,156.548
C04308=1041.917,-123.946,427.546,168.787,34.627,156.548
C04309=1041.923,-123.696,427.536,168.790,34.626,156.548
C04310=1041.929,-123.446,427.527,168.792,34.626,156.548
C04311=1041.935,-123.196,427.518,168.795,34.626,156.548
C04312=1041.941,-122.947,427.509,168.797,34.625,156.548
C04313=1041.947,-122.696,427.501,168.800,34.625,156.547
C04314=1041.954,-122.447,427.491,168.802,34.624,156.547
C04315=1041.959,-122.198,427.482,168.805,34.625,156.547
C04316=1041.965,-121.947,427.473,168.807,34.624,156.547
C04317=1041.971,-121.697,427.463,168.810,34.623,156.547
C04318=1041.978,-121.448,427.454,168.812,34.624,156.547
C04319=1041.984,-121.199,427.445,168.815,34.623,156.547
C04320=1041.990,-120.948,427.436,168.817,34.623,156.547
C04321=1041.996,-120.699,427.427,168.820,34.622,156.546
C04322=1042.002,-120.449,427.417,168.822,34.622,156.546
C04323=1042.007,-120.199,427.409,168.825,34.622,156.546
C04324=1042.014,-119.950,427.400,168.827,34.621,156.546
C04325=1042.020,-119.700,427.390,168.830,34.621,156.546
C04326=1042.026,-119.450,427.381,168.832,34.621,156.546
C04327=1042.032,-119.200,427.372,168.835,34.620,156.546
C04328=1042.038,-118.950,427.363,168.837,34.620,156.546
C04329=1042.044,-118.701,427.353,168.840,34.620,156.546
C04330=1042.050,-118.451,427.343,168.842,34.620,156.546
C04331=1042.056,-118.201,427.334,168.844,34.619,156.546
C04332=1042.063,-117.951,427.326,168.846,34.619,156.545
C04333=1042.069,-117.702,427.316,168.849,34.619,156.545
C04334=1042.075,-117.452,427.307,168.851,34.618,156.545
C04335=1042.081,-117.202,427.297,168.854,34.618,156.545
C04336=1042.087,-116.952,427.288,168.856,34.618,156.545
C04337=1042.093,-116.703,427.278,168.859,34.618,156.545
C04338=1042.099,-116.452,427.269,168.861,34.618,156.545
C04339=1042.106,-116.167,427.258,168.864,34.617,156.545
C04340=1042.113,-115.881,427.248,168.867,34.617,156.545
C04341=1042.120,-115.594,427.237,168.870,34.617,156.545
C04342=1042.127,-115.308,427.226,168.873,34.616,156.544
C04343=1042.134,-115.059,427.216,168.875,34.616,156.544
C04344=1042.139,-114.809,427.208,168.878,34.616,156.544
C04345=1042.145,-114.559,427.198,168.880,34.615,156.544
C04346=1042.151,-114.309,427.189,168.883,34.616,156.544
C04347=1042.157,-114.059,427.179,168.885,34.615,156.544
C04348=1042.164,-113.810,427.170,168.888,34.615,156.544
C04349=1042.170,-113.560,427.160,168.890,34.615,156.544
C04350=1042.176,-113.310,427.150,168.893,34.615,156.544
C04351=1042.182,-113.060,427.141,168.895,34.614,156.544
C04352=1042.188,-112.811,427.131,168.897,34.614,156.544
C04353=1042.194,-112.561,427.122,168.900,34.614,156.544
C04354=1042.199,-112.311,427.112,168.902,34.614,156.543
C04355=1042.205,-112.062,427.102,168.905,34.614,156.543
C04356=1042.212,-111.812,427.093,168.907,34.614,156.543
C04357=1042.218,-111.562,427.083,168.909,34.614,156.543
C04358=1042.224,-111.312,427.074,168.911,34.613,156.543
C04359=1042.230,-111.062,427.064,168.914,34.613,156.543
C04360=1042.237,-110.813,427.054,168.916,34.613,156.543
C04361=1042.243,-110.563,427.044,168.919,34.613,156.543
C04362=1042.249,-110.314,427.035,168.921,34.613,156.543
C04363=1042.255,-110.064,427.025,168.924,34.612,156.543
C04364=1042.261,-109.814,427.016,168.926,34.613,156.543
C04365=1042.267,-109.564,427.006,168.929,34.612,156.543
C04366=1042.274,-109.314,426.996,168.931,34.612,156.543
C04367=1042.280,-109.065,426.987,168.933,34.612,156.542
C04368=1042.285,-108.814,426.977,168.936,34.612,156.542
C04369=1042.291,-108.565,426.967,168.938,34.612,156.542
C04370=1042.298,-108.315,426.957,168.941,34.612,156.542
C04371=1042.304,-108.066,426.947,168.943,34.612,156.542
C04372=1042.310,-107.816,426.938,168.946,34.612,156.542
C04373=1042.316,-107.566,426.928,168.948,34.611,156.542
C04374=1042.323,-107.316,426.919,168.951,34.611,156.542
C04375=1042.329,-107.067,426.908,168.953,34.611,156.542
C04376=1042.334,-106.817,426.898,168.956,34.612,156.542
C04377=1042.341,-106.567,426.889,168.958,34.611,156.542
C04378=1042.347,-106.317,426.879,168.960,34.611,156.542
C04379=1042.353,-106.068,426.869,168.963,34.611,156.542
C04380=1042.359,-105.818,426.859,168.965,34.611,156.542
C04381=1042.365,-105.568,426.849,168.968,34.611,156.542
C04382=1042.371,-105.319,426.839,168.970,34.611,156.541
C04383=1042.378,-105.069,426.829,168.973,34.611,156.541
C04384=1042.383,-104.819,426.819,168.975,34.611,156.541
C04385=1042.389,-104.569,426.809,168.978,34.611,156.541
C04386=1042.395,-104.320,426.800,168.980,34.611,156.541
C04387=1042.402,-104.070,426.790,168.982,34.611,156.541
C04388=1042.407,-103.820,426.779,168.985,34.611,156.541
C04389=1042.413,-103.571,426.770,168.987,34.610,156.541
C04390=1042.420,-103.321,426.760,168.989,34.611,156.541
C04391=1042.426,-103.072,426.750,168.991,34.611,156.541
C04392=1042.431,-102.821,426.740,168.994,34.611,156.541
C04393=1042.438,-102.572,426.730,168.996,34.611,156.541
C04394=1042.444,-102.322,426.720,168.998,34.610,156.541
C04395=1042.450,-102.073,426.709,169.001,34.611,156.541
C04396=1042.457,-101.822,426.699,169.003,34.611,156.541
C04397=1042.463,-101.573,426.690,169.006,34.611,156.541
C04398=1042.469,-101.323,426.679,169.008,34.611,156.541
C04399=1042.475,-101.073,426.669,169.011,34.611,156.541
C04400=1042.481,-100.824,426.659,169.013,34.611,156.541
C04401=1042.487,-100.574,426.649,169.015,34.611,156.541
C04402=1042.493,-100.324,426.639,169.018,34.611,156.540
C04403=1042.500,-100.038,426.627,169.021,34.611,156.540
C04404=1042.507,-99.750,426.615,169.023,34.611,156.540
C04405=1042.515,-99.463,426.603,169.026,34.611,156.540
C04406=1042.522,-99.176,426.592,169.029,34.611,156.540
C04407=1042.528,-98.926,426.581,169.031,34.611,156.540
C04408=1042.534,-98.677,426.572,169.034,34.611,156.540
C04409=1042.540,-98.428,426.561,169.036,34.611,156.540
C04410=1042.546,-98.177,426.551,169.039,34.611,156.540
C04411=1042.552,-97.928,426.541,169.041,34.611,156.540
C04412=1042.559,-97.678,426.531,169.044,34.611,156.540
C04413=1042.565,-97.428,426.520,169.046,34.612,156.540
C04414=1042.571,-97.178,426.511,169.048,34.612,156.540
C04415=1042.577,-96.929,426.500,169.051,34.612,156.540
C04416=1042.583,-96.679,426.490,169.053,34.612,156.540
C04417=1042.589,-96.430,426.479,169.056,34.612,156.540
C04418=1042.596,-96.180,426.469,169.058,34.612,156.540
C04419=1042.601,-95.930,426.458,169.060,34.612,156.540
C04420=1042.607,-95.680,426.448,169.063,34.612,156.540
C04421=1042.613,-95.431,426.437,169.065,34.613,156.540
C04422=1042.619,-95.181,426.427,169.067,34.613,156.540
C04423=1042.626,-94.931,426.417,169.070,34.613,156.540
C04424=1042.632,-94.682,426.406,169.072,34.614,156.540
C04425=1042.637,-94.431,426.395,169.075,34.614,156.540
C04426=1042.643,-94.182,426.385,169.077,34.614,156.540
C04427=1042.649,-93.933,426.374,169.079,34.614,156.540
C04428=1042.656,-93.682,426.364,169.082,34.614,156.540
C04429=1042.662,-93.433,426.353,169.084,34.614,156.540
C04430=1042.667,-93.183,426.343,169.087,34.614,156.540
C04431=1042.674,-92.933,426.333,169.089,34.614,156.540
C04432=1042.679,-92.684,426.322,169.091,34.615,156.540
C04433=1042.686,-92.434,426.312,169.094,34.615,156.540
C04434=1042.692,-92.185,426.301,169.096,34.615,156.540
C04435=1042.698,-91.934,426.290,169.098,34.615,156.540
C04436=1042.704,-91.685,426.280,169.101,34.616,156.540
C04437=1042.710,-91.435,426.269,169.103,34.616,156.540
C04438=1042.717,-91.186,426.259,169.106,34.616,156.540
C04439=1042.723,-90.936,426.248,169.108,34.616,156.540
C04440=1042.729,-90.686,426.237,169.110,34.617,156.540
C04441=1042.735,-90.436,426.227,169.113,34.617,156.540
C04442=1042.741,-90.187,426.216,169.114,34.617,156.540
C04443=1042.747,-89.937,426.205,169.116,34.617,156.540
C04444=1042.754,-89.688,426.195,169.119,34.617,156.539
C04445=1042.759,-89.437,426.184,169.121,34.617,156.539
C04446=1042.766,-89.188,426.174,169.123,34.618,156.540
C04447=1042.772,-88.938,426.163,169.126,34.618,156.540
C04448=1042.778,-88.689,426.152,169.128,34.618,156.539
C04449=1042.784,-88.439,426.142,169.131,34.618,156.539
C04450=1042.790,-88.189,426.130,169.133,34.619,156.539
C04451=1042.796,-87.940,426.120,169.135,34.619,156.540
C04452=1042.803,-87.691,426.109,169.138,34.619,156.539
C04453=1042.809,-87.440,426.098,169.140,34.620,156.539
C04454=1042.814,-87.190,426.088,169.142,34.620,156.539
C04455=1042.821,-86.941,426.078,169.145,34.620,156.539
C04456=1042.827,-86.691,426.066,169.147,34.621,156.539
C04457=1042.833,-86.441,426.056,169.150,34.621,156.539
C04458=1042.840,-86.192,426.045,169.152,34.621,156.539
C04459=1042.846,-85.942,426.034,169.154,34.621,156.539
C04460=1042.852,-85.693,426.023,169.157,34.621,156.539
C04461=1042.859,-85.443,426.012,169.159,34.622,156.539
C04462=1042.864,-85.193,426.002,169.161,34.622,156.539
C04463=1042.871,-84.943,425.990,169.164,34.622,156.539
C04464=1042.877,-84.694,425.980,169.166,34.622,156.539
C04465=1042.883,-84.444,425.969,169.168,34.623,156.539
C04466=1042.889,-84.194,425.958,169.171,34.623,156.539
C04467=1042.896,-83.910,425.946,169.173,34.623,156.539
C04468=1042.904,-83.625,425.933,169.176,34.623,156.539
C04469=1042.911,-83.339,425.921,169.179,34.624,156.539
C04470=1042.918,-83.055,425.908,169.181,34.624,156.539
C04471=1042.925,-82.806,425.897,169.184,34.624,156.539
C04472=1042.931,-82.556,425.887,169.186,34.625,156.539
C04473=1042.937,-82.307,425.876,169.189,34.625,156.539
C04474=1042.943,-82.056,425.864,169.191,34.625,156.539
C04475=1042.949,-81.807,425.854,169.193,34.625,156.539
C04476=1042.956,-81.557,425.843,169.196,34.626,156.539
C04477=1042.961,-81.308,425.832,169.198,34.626,156.539
C04478=1042.969,-81.058,425.821,169.200,34.626,156.539
C04479=1042.974,-80.808,425.810,169.203,34.627,156.539
C04480=1042.981,-80.559,425.799,169.205,34.627,156.539
C04481=1042.987,-80.309,425.788,169.207,34.627,156.539
C04482=1042.994,-80.059,425.777,169.210,34.628,156.539
C04483=1043.000,-79.809,425.766,169.212,34.628,156.540
C04484=1043.006,-79.560,425.755,169.214,34.628,156.539
C04485=1043.012,-79.309,425.744,169.217,34.629,156.540
C04486=1043.018,-79.060,425.732,169.219,34.629,156.540
C04487=1043.025,-78.810,425.721,169.221,34.629,156.540
C04488=1043.030,-78.561,425.710,169.224,34.630,156.540
C04489=1043.037,-78.311,425.699,169.226,34.630,156.540
C04490=1043.043,-78.062,425.687,169.228,34.631,156.540
C04491=1043.049,-77.812,425.676,169.230,34.631,156.540
C04492=1043.056,-77.562,425.666,169.233,34.632,156.540
C04493=1043.062,-77.312,425.654,169.235,34.632,156.540
C04494=1043.068,-77.063,425.643,169.237,34.633,156.540
C04495=1043.074,-76.813,425.631,169.240,34.633,156.540
C04496=1043.080,-76.564,425.621,169.242,34.634,156.540
C04497=1043.087,-76.314,425.609,169.244,34.634,156.540
C04498=1043.092,-76.065,425.598,169.247,34.635,156.540
C04499=1043.099,-75.814,425.587,169.249,34.635,156.540
C04500=1043.105,-75.565,425.575,169.251,34.635,156.540
C04501=1043.111,-75.315,425.564,169.253,34.635,156.540
C04502=1043.117,-75.065,425.552,169.256,34.636,156.540
C04503=1043.123,-74.816,425.541,169.258,34.636,156.540
C04504=1043.130,-74.566,425.530,169.260,34.637,156.540
C04505=1043.136,-74.317,425.519,169.263,34.637,156.540
C04506=1043.142,-74.067,425.507,169.265,34.638,156.540
C04507=1043.148,-73.817,425.496,169.267,34.639,156.540
C04508=1043.155,-73.568,425.484,169.269,34.639,156.540
C04509=1043.160,-73.317,425.472,169.272,34.640,156.540
C04510=1043.166,-73.069,425.460,169.274,34.640,156.540
C04511=1043.173,-72.818,425.449,169.276,34.640,156.540
C04512=1043.178,-72.569,425.438,169.279,34.641,156.540
C04513=1043.185,-72.319,425.426,169.281,34.642,156.540
C04514=1043.190,-72.069,425.415,169.283,34.642,156.540
C04515=1043.197,-71.820,425.403,169.285,34.643,156.541
C04516=1043.203,-71.570,425.391,169.288,34.644,156.541
C04517=1043.209,-71.321,425.380,169.290,34.644,156.541
C04518=1043.215,-71.071,425.368,169.292,34.644,156.541
C04519=1043.221,-70.821,425.357,169.294,34.645,156.541
C04520=1043.227,-70.572,425.345,169.297,34.646,156.541
C04521=1043.234,-70.322,425.334,169.299,34.647,156.541
C04522=1043.239,-70.073,425.321,169.301,34.647,156.541
C04523=1043.245,-69.822,425.310,169.303,34.648,156.541
C04524=1043.251,-69.573,425.298,169.306,34.648,156.541
C04525=1043.258,-69.324,425.287,169.308,34.648,156.541
C04526=1043.264,-69.073,425.275,169.310,34.649,156.541
C04527=1043.270,-68.825,425.263,169.312,34.650,156.541
C04528=1043.276,-68.574,425.252,169.315,34.651,156.541
C04529=1043.283,-68.325,425.240,169.317,34.651,156.541
C04530=1043.288,-68.076,425.228,169.319,34.652,156.541
C04531=1043.295,-67.792,425.214,169.322,34.652,156.541
C04532=1043.302,-67.510,425.201,169.324,34.653,156.542
C04533=1043.309,-67.227,425.188,169.327,34.654,156.542
C04534=1043.316,-66.945,425.175,169.329,34.655,156.542
C04535=1043.322,-66.695,425.163,169.331,34.655,156.542
C04536=1043.328,-66.446,425.152,169.334,34.656,156.542
C04537=1043.334,-66.196,425.139,169.336,34.656,156.542
C04538=1043.341,-65.946,425.127,169.338,34.657,156.542
C04539=1043.347,-65.696,425.116,169.340,34.658,156.542
C04540=1043.353,-65.447,425.104,169.343,34.658,156.542
C04541=1043.359,-65.197,425.092,169.345,34.659,156.542
C04542=1043.366,-64.948,425.080,169.347,34.659,156.542
C04543=1043.372,-64.698,425.069,169.349,34.660,156.542
C04544=1043.377,-64.448,425.056,169.352,34.661,156.542
C04545=1043.384,-64.199,425.045,169.354,34.661,156.542
C04546=1043.391,-63.949,425.033,169.356,34.662,156.542
C04547=1043.397,-63.699,425.021,169.358,34.662,156.543
C04548=1043.402,-63.450,425.009,169.361,34.663,156.543
C04549=1043.409,-63.200,424.997,169.363,34.664,156.543
C04550=1043.416,-62.951,424.985,169.365,34.664,156.543
C04551=1043.421,-62.701,424.973,169.367,34.665,156.543
C04552=1043.427,-62.451,424.962,169.369,34.666,156.543
C04553=1043.434,-62.202,424.950,169.372,34.666,156.543
C04554=1043.440,-61.952,424.937,169.374,34.667,156.543
C04555=1043.446,-61.702,424.925,169.376,34.667,156.543
C04556=1043.453,-61.453,424.913,169.378,34.668,156.543
C04557=1043.458,-61.204,424.901,169.381,34.669,156.543
C04558=1043.465,-60.953,424.890,169.383,34.669,156.543
C04559=1043.471,-60.704,424.878,169.385,34.670,156.543
C04560=1043.477,-60.454,424.865,169.387,34.671,156.543
C04561=1043.484,-60.204,424.853,169.389,34.671,156.543
C04562=1043.491,-59.955,424.841,169.392,34.672,156.543
C04563=1043.496,-59.706,424.829,169.394,34.673,156.544
C04564=1043.503,-59.456,424.817,169.396,34.673,156.544
C04565=1043.509,-59.206,424.805,169.398,34.674,156.544
C04566=1043.515,-58.957,424.793,169.401,34.675,156.544
C04567=1043.522,-58.707,424.781,169.403,34.675,156.544
C04568=1043.528,-58.457,424.769,169.405,34.676,156.544
C04569=1043.534,-58.207,424.757,169.407,34.676,156.544
C04570=1043.540,-57.958,424.745,169.409,34.677,156.544
C04571=1043.547,-57.708,424.734,169.412,34.678,156.544
C04572=1043.553,-57.459,424.721,169.415,34.679,156.544
C04573=1043.559,-57.209,424.709,169.417,34.679,156.544
C04574=1043.566,-56.959,424.697,169.419,34.680,156.544
C04575=1043.572,-56.710,424.685,169.421,34.681,156.544
C04576=1043.578,-56.460,424.673,169.424,34.681,156.544
C04577=1043.584,-56.210,424.660,169.426,34.682,156.545
C04578=1043.591,-55.961,424.648,169.428,34.682,156.545
C04579=1043.598,-55.711,424.636,169.430,34.683,156.545
C04580=1043.604,-55.462,424.623,169.432,34.684,156.545
C04581=1043.610,-55.212,424.611,169.435,34.685,156.545
C04582=1043.617,-54.963,424.599,169.437,34.685,156.545
C04583=1043.622,-54.713,424.587,169.439,34.686,156.545
C04584=1043.629,-54.464,424.575,169.441,34.686,156.545
C04585=1043.635,-54.214,424.562,169.443,34.687,156.545
C04586=1043.642,-53.964,424.550,169.446,34.688,156.545
C04587=1043.648,-53.715,424.538,169.448,34.688,156.545
C04588=1043.654,-53.465,424.526,169.450,34.689,156.545
C04589=1043.661,-53.215,424.514,169.452,34.690,156.545
C04590=1043.667,-52.965,424.501,169.454,34.691,156.546
C04591=1043.674,-52.716,424.489,169.457,34.691,156.546
C04592=1043.680,-52.467,424.477,169.459,34.692,156.546
C04593=1043.686,-52.217,424.464,169.461,34.693,156.546
C04594=1043.693,-51.967,424.452,169.463,34.694,156.546
C04595=1043.700,-51.686,424.438,169.466,34.694,156.546
C04596=1043.707,-51.404,424.424,169.468,34.695,156.546
C04597=1043.714,-51.123,424.410,169.470,34.696,156.546
C04598=1043.722,-50.842,424.396,169.473,34.697,156.546
C04599=1043.728,-50.592,424.383,169.475,34.697,156.546
C04600=1043.735,-50.343,424.371,169.477,34.698,156.546
C04601=1043.741,-50.093,424.359,169.479,34.699,156.547
C04602=1043.747,-49.843,424.346,169.482,34.700,156.547
C04603=1043.753,-49.594,424.333,169.484,34.700,156.547
C04604=1043.759,-49.344,424.321,169.486,34.701,156.547
C04605=1043.765,-49.094,424.309,169.488,34.703,156.547
C04606=1043.772,-48.845,424.295,169.490,34.703,156.547
C04607=1043.778,-48.595,424.283,169.492,34.704,156.547
C04608=1043.784,-48.346,424.271,169.494,34.705,156.547
C04609=1043.790,-48.096,424.258,169.496,34.705,156.547
C04610=1043.796,-47.846,424.245,169.499,34.706,156.547
C04611=1043.803,-47.597,424.233,169.501,34.708,156.548
C04612=1043.809,-47.348,424.220,169.503,34.708,156.548
C04613=1043.815,-47.098,424.207,169.505,34.709,156.548
C04614=1043.821,-46.848,424.194,169.507,34.710,156.548
C04615=1043.827,-46.599,424.181,169.509,34.711,156.548
C04616=1043.834,-46.349,424.169,169.511,34.711,156.548
C04617=1043.840,-46.100,424.156,169.514,34.713,156.548
C04618=1043.846,-45.849,424.143,169.516,34.713,156.548
C04619=1043.853,-45.600,424.130,169.518,34.714,156.548
C04620=1043.859,-45.350,424.118,169.520,34.715,156.549
C04621=1043.865,-45.100,424.105,169.522,34.716,156.549
C04622=1043.871,-44.851,424.092,169.524,34.717,156.549
C04623=1043.877,-44.601,424.080,169.526,34.718,156.549
C04624=1043.884,-44.352,424.067,169.528,34.718,156.549
C04625=1043.890,-44.102,424.054,169.530,34.719,156.549
C04626=1043.896,-43.853,424.041,169.534,34.720,156.549
C04627=1043.902,-43.603,424.029,169.536,34.721,156.549
C04628=1043.909,-43.354,424.015,169.538,34.722,156.550
C04629=1043.916,-43.104,424.003,169.540,34.723,156.550
C04630=1043.922,-42.854,423.990,169.542,34.724,156.550
C04631=1043.928,-42.605,423.977,169.544,34.724,156.550
C04632=1043.934,-42.355,423.964,169.546,34.726,156.550
C04633=1043.940,-42.105,423.951,169.548,34.726,156.550
C04634=1043.947,-41.856,423.939,169.550,34.727,156.550
C04635=1043.953,-41.607,423.926,169.553,34.728,156.550
C04636=1043.960,-41.357,423.912,169.555,34.729,156.550
C04637=1043.966,-41.107,423.899,169.557,34.730,156.551
C04638=1043.972,-40.857,423.887,169.559,34.731,156.551
C04639=1043.979,-40.609,423.874,169.561,34.731,156.551
C04640=1043.985,-40.359,423.861,169.563,34.732,156.551
C04641=1043.991,-40.109,423.848,169.565,34.733,156.551
C04642=1043.998,-39.859,423.835,169.567,34.734,156.551
C04643=1044.004,-39.610,423.822,169.569,34.735,156.551
C04644=1044.010,-39.360,423.809,169.572,34.736,156.551
C04645=1044.016,-39.111,423.797,169.574,34.737,156.551
C04646=1044.023,-38.861,423.783,169.576,34.738,156.552
C04647=1044.030,-38.611,423.770,169.578,34.739,156.552
C04648=1044.035,-38.362,423.757,169.580,34.739,156.552
C04649=1044.042,-38.112,423.744,169.582,34.741,156.552
C04650=1044.048,-37.863,423.731,169.584,34.741,156.552
C04651=1044.054,-37.613,423.718,169.586,34.743,156.552
C04652=1044.061,-37.363,423.705,169.588,34.743,156.552
C04653=1044.067,-37.114,423.691,169.590,34.744,156.552
C04654=1044.072,-36.864,423.677,169.592,34.746,156.553
C04655=1044.078,-36.614,423.665,169.594,34.746,156.553
C04656=1044.084,-36.365,423.652,169.596,34.748,156.553
C04657=1044.091,-36.115,423.638,169.598,34.748,156.553
C04658=1044.097,-35.866,423.625,169.600,34.749,156.553
C04659=1044.104,-35.585,423.611,169.603,34.751,156.553
C04660=1044.112,-35.304,423.595,169.606,34.751,156.553
C04661=1044.118,-35.024,423.580,169.608,34.753,156.554
C04662=1044.126,-34.743,423.566,169.611,34.754,156.554
C04663=1044.132,-34.493,423.552,169.613,34.755,156.554
C04664=1044.139,-34.243,423.539,169.615,34.755,156.554
C04665=1044.145,-33.994,423.526,169.617,34.757,156.554
C04666=1044.151,-33.744,423.513,169.619,34.758,156.554
C04667=1044.156,-33.495,423.499,169.621,34.759,156.554
C04668=1044.163,-33.245,423.485,169.623,34.760,156.555
C04669=1044.169,-32.995,423.472,169.625,34.761,156.555
C04670=1044.175,-32.746,423.459,169.627,34.762,156.555
C04671=1044.182,-32.497,423.446,169.629,34.762,156.555
C04672=1044.188,-32.247,423.432,169.631,34.764,156.555
C04673=1044.195,-31.998,423.419,169.633,34.765,156.555
C04674=1044.201,-31.748,423.406,169.635,34.766,156.555
C04675=1044.207,-31.498,423.393,169.637,34.767,156.556
C04676=1044.214,-31.249,423.379,169.639,34.767,156.556
C04677=1044.220,-30.999,423.366,169.641,34.769,156.556
C04678=1044.226,-30.749,423.352,169.643,34.769,156.556
C04679=1044.232,-30.500,423.339,169.646,34.771,156.556
C04680=1044.238,-30.251,423.325,169.648,34.772,156.556
C04681=1044.245,-30.001,423.312,169.650,34.773,156.556
C04682=1044.251,-29.751,423.298,169.652,34.774,156.557
C04683=1044.258,-29.502,423.285,169.654,34.774,156.557
C04684=1044.264,-29.252,423.271,169.656,34.776,156.557
C04685=1044.271,-29.003,423.258,169.658,34.776,156.557
C04686=1044.277,-28.754,423.245,169.660,34.778,156.557
C04687=1044.283,-28.503,423.231,169.662,34.779,156.557
C04688=1044.289,-28.254,423.217,169.665,34.780,156.557
C04689=1044.296,-28.004,423.204,169.667,34.781,156.558
C04690=1044.302,-27.755,423.190,169.669,34.782,156.558
C04691=1044.308,-27.506,423.177,169.671,34.783,156.558
C04692=1044.315,-27.256,423.164,169.673,34.783,156.558
C04693=1044.321,-27.006,423.150,169.675,34.785,156.558
C04694=1044.327,-26.756,423.136,169.677,34.786,156.558
C04695=1044.334,-26.507,423.123,169.679,34.787,156.558
C04696=1044.340,-26.258,423.109,169.681,34.788,156.559
C04697=1044.346,-26.008,423.095,169.683,34.789,156.559
C04698=1044.352,-25.759,423.081,169.685,34.790,156.559
C04699=1044.359,-25.509,423.068,169.687,34.791,156.559
C04700=1044.365,-25.259,423.054,169.689,34.792,156.559
C04701=1044.371,-25.010,423.041,169.691,34.794,156.559
C04702=1044.376,-24.760,423.027,169.693,34.795,156.560
C04703=1044.384,-24.511,423.012,169.695,34.796,156.560
C04704=1044.390,-24.262,422.999,169.697,34.797,156.560
C04705=1044.396,-24.011,422.985,169.699,34.798,156.560
C04706=1044.402,-23.762,422.972,169.701,34.799,156.560
C04707=1044.409,-23.512,422.958,169.703,34.800,156.560
C04708=1044.415,-23.263,422.943,169.705,34.801,156.561
C04709=1044.421,-23.014,422.930,169.707,34.802,156.561
C04710=1044.427,-22.764,422.916,169.709,34.803,156.561
C04711=1044.433,-22.514,422.903,169.712,34.805,156.561
C04712=1044.440,-22.265,422.888,169.714,34.806,156.561
C04713=1044.446,-22.015,422.874,169.716,34.807,156.561
C04714=1044.453,-21.765,422.861,169.718,34.808,156.561
C04715=1044.458,-21.516,422.847,169.720,34.809,156.562
C04716=1044.465,-21.267,422.833,169.722,34.810,156.562
C04717=1044.471,-21.017,422.819,169.724,34.811,156.562
C04718=1044.477,-20.768,422.805,169.726,34.812,156.562
C04719=1044.484,-20.518,422.791,169.728,34.814,156.562
C04720=1044.490,-20.269,422.778,169.730,34.815,156.562
C04721=1044.496,-20.019,422.764,169.731,34.816,156.563
C04722=1044.502,-19.770,422.750,169.733,34.817,156.563
C04723=1044.510,-19.488,422.734,169.736,34.818,156.563
C04724=1044.517,-19.207,422.718,169.738,34.819,156.563
C04725=1044.524,-18.925,422.702,169.740,34.821,156.563
C04726=1044.532,-18.642,422.687,169.742,34.822,156.564
C04727=1044.537,-18.417,422.674,169.744,34.823,156.564
C04728=1044.542,-18.191,422.661,169.746,34.824,156.564
C04729=1044.549,-17.965,422.649,169.748,34.825,156.564
C04730=1044.554,-17.739,422.636,169.749,34.826,156.564
C04731=1044.560,-17.514,422.624,169.751,34.827,156.564
C04732=1044.565,-17.288,422.611,169.753,34.828,156.564
C04733=1044.572,-17.062,422.599,169.756,34.829,156.565
C04734=1044.577,-16.837,422.585,169.758,34.830,156.565
C04735=1044.583,-16.587,422.571,169.759,34.831,156.565
C04736=1044.590,-16.337,422.557,169.761,34.832,156.565
C04737=1044.597,-16.088,422.543,169.763,34.833,156.565
C04738=1044.602,-15.838,422.529,169.765,34.834,156.565
C04739=1044.609,-15.589,422.515,169.767,34.836,156.566
C04740=1044.615,-15.339,422.501,169.769,34.836,156.566
C04741=1044.622,-15.090,422.487,169.771,34.838,156.566
C04742=1044.627,-14.840,422.473,169.773,34.839,156.566
C04743=1044.634,-14.591,422.458,169.775,34.841,156.566
C04744=1044.640,-14.341,422.445,169.777,34.841,156.566
C04745=1044.646,-14.092,422.430,169.779,34.843,156.567
C04746=1044.653,-13.841,422.415,169.781,34.844,156.567
C04747=1044.659,-13.593,422.401,169.783,34.845,156.567
C04748=1044.665,-13.343,422.386,169.785,34.846,156.567
C04749=1044.671,-13.094,422.373,169.787,34.847,156.567
C04750=1044.678,-12.844,422.358,169.789,34.849,156.568
C04751=1044.684,-12.595,422.344,169.790,34.850,156.568
C04752=1044.690,-12.345,422.329,169.792,34.851,156.568
C04753=1044.697,-12.095,422.316,169.795,34.852,156.568
C04754=1044.703,-11.846,422.301,169.797,34.853,156.568
C04755=1044.709,-11.596,422.286,169.799,34.855,156.568
C04756=1044.715,-11.347,422.273,169.801,34.856,156.569
C04757=1044.721,-11.098,422.258,169.803,34.857,156.569
C04758=1044.728,-10.848,422.243,169.805,34.858,156.569
C04759=1044.734,-10.599,422.230,169.807,34.860,156.569
C04760=1044.740,-10.349,422.215,169.809,34.861,156.569
C04761=1044.747,-10.099,422.200,169.811,34.862,156.570
C04762=1044.753,-9.850,422.187,169.812,34.863,156.570
C04763=1044.759,-9.600,422.172,169.814,34.864,156.570
C04764=1044.765,-9.351,422.157,169.816,34.866,156.570
C04765=1044.771,-9.101,422.143,169.818,34.867,156.570
C04766=1044.778,-8.852,422.129,169.820,34.868,156.571
C04767=1044.784,-8.603,422.114,169.822,34.869,156.571
C04768=1044.791,-8.353,422.099,169.824,34.870,156.571
C04769=1044.797,-8.103,422.085,169.826,34.872,156.571
C04770=1044.803,-7.854,422.071,169.828,34.873,156.571
C04771=1044.810,-7.605,422.056,169.831,34.874,156.571
C04772=1044.816,-7.355,422.041,169.833,34.875,156.572
C04773=1044.823,-7.105,422.027,169.834,34.876,156.572
C04774=1044.829,-6.856,422.013,169.836,34.878,156.572
C04775=1044.835,-6.606,421.998,169.838,34.879,156.572
C04776=1044.842,-6.357,421.983,169.840,34.880,156.572
C04777=1044.848,-6.107,421.970,169.842,34.881,156.572
C04778=1044.854,-5.858,421.955,169.844,34.883,156.573
C04779=1044.860,-5.608,421.940,169.846,34.884,156.573
C04780=1044.867,-5.359,421.925,169.848,34.885,156.573
C04781=1044.873,-5.110,421.911,169.850,34.886,156.573
C04782=1044.879,-4.860,421.897,169.851,34.887,156.573
C04783=1044.886,-4.610,421.882,169.853,34.889,156.574
C04784=1044.893,-4.361,421.867,169.855,34.890,156.574
C04785=1044.899,-4.112,421.853,169.857,34.891,156.574
C04786=1044.905,-3.862,421.838,169.859,34.892,156.574
C04787=1044.914,-3.531,421.819,169.862,34.894,156.574
C04788=1044.922,-3.201,421.799,169.864,34.895,156.575
C04789=1044.930,-2.869,421.779,169.867,34.897,156.575
C04790=1044.938,-2.539,421.759,169.870,34.899,156.575
C04791=1044.944,-2.289,421.744,169.872,34.901,156.576
C04792=1044.951,-2.040,421.729,169.874,34.902,156.576
C04793=1044.956,-1.791,421.715,169.875,34.903,156.576
C04794=1044.963,-1.541,421.700,169.877,34.905,156.576
C04795=1044.969,-1.291,421.685,169.879,34.906,156.576
C04796=1044.976,-1.042,421.670,169.881,34.907,156.577
C04797=1044.981,-0.793,421.655,169.883,34.909,156.577
C04798=1044.988,-0.543,421.641,169.885,34.910,156.577
C04799=1044.994,-0.293,421.626,169.886,34.911,156.577
C04800=1045.000,-0.044,421.611,169.888,34.912,156.577
C04801=1045.006,0.205,421.596,169.890,34.914,156.578
C04802=1045.013,0.455,421.581,169.892,34.915,156.578
C04803=1045.019,0.704,421.566,169.894,34.916,156.578
C04804=1045.025,0.954,421.551,169.897,34.918,156.578
C04805=1045.031,1.203,421.537,169.899,34.919,156.578
C04806=1045.038,1.453,421.522,169.900,34.920,156.579
C04807=1045.044,1.702,421.507,169.902,34.922,156.579
C04808=1045.050,1.952,421.491,169.904,34.923,156.579
C04809=1045.056,2.201,421.476,169.906,34.924,156.579
C04810=1045.062,2.450,421.461,169.908,34.926,156.579
C04811=1045.068,2.700,421.446,169.910,34.927,156.580
C04812=1045.075,2.950,421.431,169.911,34.928,156.580
C04813=1045.081,3.199,421.416,169.913,34.930,156.580
C04814=1045.088,3.449,421.401,169.915,34.931,156.580
C04815=1045.093,3.698,421.387,169.917,34.932,156.580
C04816=1045.100,3.948,421.372,169.919,34.934,156.581
C04817=1045.106,4.197,421.356,169.921,34.935,156.581
C04818=1045.113,4.446,421.341,169.922,34.936,156.581
C04819=1045.119,4.696,421.326,169.925,34.938,156.581
C04820=1045.126,4.946,421.311,169.927,34.939,156.582
C04821=1045.131,5.196,421.296,169.929,34.940,156.582
C04822=1045.137,5.444,421.280,169.931,34.942,156.582
C04823=1045.144,5.694,421.265,169.932,34.943,156.582
C04824=1045.150,5.943,421.250,169.934,34.944,156.582
C04825=1045.156,6.193,421.235,169.936,34.946,156.583
C04826=1045.163,6.443,421.221,169.938,34.947,156.583
C04827=1045.170,6.692,421.205,169.940,34.948,156.583
C04828=1045.176,6.941,421.190,169.942,34.950,156.583
C04829=1045.182,7.191,421.175,169.943,34.951,156.583
C04830=1045.189,7.440,421.159,169.945,34.952,156.584
C04831=1045.194,7.689,421.144,169.947,34.954,156.584
C04832=1045.200,7.939,421.129,169.949,34.955,156.584
C04833=1045.207,8.189,421.114,169.952,34.956,156.584
C04834=1045.213,8.438,421.099,169.954,34.958,156.584
C04835=1045.220,8.687,421.084,169.955,34.959,156.585
C04836=1045.226,8.937,421.069,169.957,34.960,156.585
C04837=1045.233,9.186,421.053,169.959,34.962,156.585
C04838=1045.239,9.436,421.038,169.961,34.963,156.585
C04839=1045.245,9.686,421.023,169.963,34.964,156.586
C04840=1045.252,9.935,421.007,169.964,34.966,156.586
C04841=1045.258,10.184,420.992,169.966,34.967,156.586
C04842=1045.264,10.434,420.977,169.968,34.968,156.586
C04843=1045.271,10.683,420.961,169.970,34.970,156.586
C04844=1045.277,10.933,420.946,169.972,34.971,156.587
C04845=1045.284,11.182,420.931,169.973,34.972,156.587
C04846=1045.290,11.432,420.915,169.975,34.974,156.587
C04847=1045.296,11.681,420.900,169.977,34.975,156.587
C04848=1045.303,11.930,420.885,169.980,34.976,156.587
C04849=1045.309,12.180,420.870,169.982,34.978,156.588
C04850=1045.316,12.430,420.855,169.984,34.979,156.588
C04851=1045.323,12.714,420.837,169.986,34.980,156.588
C04852=1045.330,12.999,420.820,169.988,34.982,156.588
C04853=1045.338,13.285,420.802,169.990,34.983,156.589
C04854=1045.345,13.570,420.784,169.992,34.985,156.589
C04855=1045.351,13.820,420.769,169.994,34.986,156.589
C04856=1045.358,14.069,420.753,169.995,34.988,156.589
C04857=1045.364,14.318,420.738,169.997,34.989,156.590
C04858=1045.371,14.567,420.723,169.999,34.990,156.590
C04859=1045.376,14.817,420.707,170.001,34.992,156.590
C04860=1045.383,15.066,420.691,170.002,34.993,156.590
C04861=1045.389,15.316,420.676,170.004,34.994,156.590
C04862=1045.395,15.565,420.660,170.007,34.996,156.591
C04863=1045.402,15.814,420.644,170.009,34.997,156.591
C04864=1045.408,16.064,420.629,170.011,34.998,156.591
C04865=1045.414,16.313,420.613,170.012,35.000,156.591
C04866=1045.420,16.563,420.598,170.014,35.001,156.592
C04867=1045.427,16.812,420.582,170.016,35.003,156.592
C04868=1045.433,17.062,420.567,170.018,35.004,156.592
C04869=1045.439,17.311,420.551,170.019,35.005,156.592
C04870=1045.446,17.561,420.535,170.021,35.007,156.592
C04871=1045.451,17.811,420.520,170.023,35.008,156.593
C04872=1045.458,18.060,420.504,170.025,35.009,156.593
C04873=1045.465,18.309,420.488,170.027,35.011,156.593
C04874=1045.470,18.559,420.473,170.028,35.013,156.593
C04875=1045.477,18.808,420.457,170.031,35.014,156.594
C04876=1045.484,19.058,420.441,170.033,35.015,156.594
C04877=1045.490,19.307,420.426,170.035,35.017,156.594
C04878=1045.497,19.556,420.410,170.036,35.018,156.594
C04879=1045.503,19.806,420.394,170.038,35.019,156.594
C04880=1045.509,20.055,420.379,170.040,35.021,156.595
C04881=1045.515,20.305,420.362,170.042,35.022,156.595
C04882=1045.522,20.554,420.347,170.043,35.024,156.595
C04883=1045.527,20.804,420.331,170.045,35.025,156.595
C04884=1045.534,21.053,420.316,170.047,35.027,156.596
C04885=1045.540,21.302,420.299,170.049,35.028,156.596
C04886=1045.546,21.551,420.283,170.050,35.029,156.596
C04887=1045.552,21.801,420.268,170.052,35.031,156.596
C04888=1045.559,22.051,420.251,170.055,35.032,156.597
C04889=1045.565,22.300,420.236,170.057,35.034,156.597
C04890=1045.571,22.550,420.220,170.058,35.035,156.597
C04891=1045.578,22.799,420.204,170.060,35.036,156.597
C04892=1045.584,23.049,420.188,170.062,35.038,156.597
C04893=1045.590,23.298,420.173,170.064,35.040,156.598
C04894=1045.596,23.547,420.156,170.065,35.041,156.598
C04895=1045.602,23.796,420.140,170.067,35.042,156.598
C04896=1045.610,24.046,420.124,170.069,35.044,156.598
C04897=1045.615,24.296,420.109,170.071,35.045,156.599
C04898=1045.622,24.545,420.093,170.072,35.046,156.599
C04899=1045.628,24.794,420.077,170.074,35.048,156.599
C04900=1045.635,25.043,420.061,170.077,35.050,156.599
C04901=1045.641,25.293,420.045,170.079,35.051,156.600
C04902=1045.647,25.542,420.029,170.080,35.052,156.600
C04903=1045.654,25.792,420.013,170.082,35.054,156.600
C04904=1045.660,26.041,419.996,170.084,35.055,156.600
C04905=1045.666,26.291,419.981,170.085,35.057,156.601
C04906=1045.672,26.540,419.965,170.087,35.058,156.601
C04907=1045.678,26.790,419.949,170.089,35.059,156.601
C04908=1045.685,27.039,419.933,170.091,35.061,156.601
C04909=1045.691,27.289,419.917,170.092,35.062,156.601
C04910=1045.698,27.538,419.901,170.094,35.063,156.602
C04911=1045.704,27.787,419.885,170.096,35.065,156.602
C04912=1045.710,28.036,419.868,170.098,35.067,156.602
C04913=1045.717,28.285,419.853,170.100,35.068,156.602
C04914=1045.723,28.535,419.836,170.102,35.069,156.603
C04915=1045.731,28.822,419.817,170.104,35.071,156.603
C04916=1045.737,29.109,419.799,170.106,35.073,156.603
C04917=1045.744,29.395,419.780,170.108,35.075,156.604
C04918=1045.752,29.681,419.762,170.110,35.077,156.604
C04919=1045.758,29.931,419.745,170.112,35.078,156.604
C04920=1045.764,30.180,419.729,170.113,35.079,156.604
C04921=1045.770,30.429,419.713,170.115,35.080,156.605
C04922=1045.776,30.678,419.697,170.117,35.082,156.605
C04923=1045.783,30.928,419.681,170.119,35.084,156.605
C04924=1045.789,31.178,419.664,170.121,35.085,156.605
C04925=1045.795,31.427,419.647,170.123,35.087,156.606
C04926=1045.802,31.676,419.632,170.125,35.088,156.606
C04927=1045.808,31.926,419.615,170.126,35.090,156.606
C04928=1045.814,32.175,419.599,170.128,35.091,156.606
C04929=1045.820,32.424,419.583,170.130,35.093,156.607
C04930=1045.826,32.674,419.566,170.131,35.094,156.607
C04931=1045.833,32.924,419.550,170.133,35.096,156.607
C04932=1045.839,33.173,419.534,170.135,35.097,156.607
C04933=1045.846,33.421,419.517,170.137,35.099,156.608
C04934=1045.852,33.671,419.501,170.138,35.100,156.608
C04935=1045.858,33.921,419.484,170.141,35.101,156.608
C04936=1045.864,34.170,419.468,170.143,35.103,156.608
C04937=1045.871,34.419,419.452,170.144,35.105,156.609
C04938=1045.877,34.669,419.436,170.146,35.106,156.609
C04939=1045.884,34.918,419.419,170.148,35.107,156.609
C04940=1045.889,35.167,419.402,170.150,35.109,156.609
C04941=1045.895,35.417,419.386,170.151,35.111,156.610
C04942=1045.902,35.667,419.369,170.153,35.112,156.610
C04943=1045.909,35.916,419.354,170.155,35.113,156.610
C04944=1045.915,36.165,419.337,170.156,35.114,156.610
C04945=1045.921,36.415,419.320,170.158,35.116,156.611
C04946=1045.927,36.664,419.304,170.160,35.118,156.611
C04947=1045.933,36.913,419.288,170.163,35.119,156.611
C04948=1045.940,37.163,419.270,170.164,35.120,156.611
C04949=1045.946,37.412,419.254,170.166,35.122,156.612
C04950=1045.953,37.661,419.238,170.168,35.124,156.612
C04951=1045.960,37.911,419.221,170.169,35.125,156.612
C04952=1045.965,38.160,419.204,170.171,35.127,156.612
C04953=1045.971,38.410,419.188,170.173,35.128,156.612
C04954=1045.977,38.658,419.171,170.174,35.130,156.613
C04955=1045.984,38.908,419.154,170.176,35.131,156.613
C04956=1045.990,39.158,419.138,170.178,35.133,156.613
C04957=1045.996,39.406,419.121,170.179,35.134,156.613
C04958=1046.002,39.656,419.105,170.182,35.136,156.614
C04959=1046.008,39.906,419.088,170.184,35.137,156.614
C04960=1046.015,40.155,419.071,170.185,35.139,156.614
C04961=1046.021,40.405,419.055,170.187,35.141,156.615
C04962=1046.027,40.653,419.038,170.189,35.142,156.615
C04963=1046.033,40.903,419.021,170.191,35.143,156.615
C04964=1046.040,41.153,419.005,170.192,35.145,156.615
C04965=1046.046,41.401,418.988,170.194,35.146,156.616
C04966=1046.053,41.652,418.971,170.196,35.148,156.616
C04967=1046.059,41.900,418.954,170.197,35.150,156.616
C04968=1046.065,42.150,418.938,170.200,35.151,156.616
C04969=1046.071,42.399,418.920,170.202,35.153,156.617
C04970=1046.077,42.649,418.904,170.203,35.154,156.617
C04971=1046.083,42.898,418.888,170.205,35.156,156.617
C04972=1046.090,43.147,418.870,170.207,35.158,156.617
C04973=1046.096,43.397,418.854,170.208,35.159,156.618
C04974=1046.103,43.646,418.837,170.210,35.160,156.618
C04975=1046.109,43.896,418.820,170.212,35.162,156.618
C04976=1046.114,44.145,418.803,170.213,35.163,156.618
C04977=1046.121,44.394,418.786,170.215,35.165,156.619
C04978=1046.127,44.643,418.769,170.217,35.167,156.619
C04979=1046.134,44.929,418.749,170.220,35.169,156.619
C04980=1046.141,45.217,418.730,170.221,35.170,156.620
C04981=1046.148,45.503,418.710,170.223,35.172,156.620
C04982=1046.155,45.789,418.691,170.225,35.174,156.620
C04983=1046.161,46.038,418.674,170.227,35.176,156.621
C04984=1046.168,46.288,418.657,170.229,35.177,156.621
C04985=1046.173,46.537,418.639,170.230,35.179,156.621
C04986=1046.180,46.787,418.623,170.232,35.180,156.621
C04987=1046.186,47.036,418.606,170.233,35.182,156.622
C04988=1046.191,47.285,418.588,170.236,35.183,156.622
C04989=1046.198,47.535,418.572,170.238,35.185,156.622
C04990=1046.204,47.784,418.555,170.239,35.187,156.622
C04991=1046.210,48.034,418.537,170.241,35.189,156.623
C04992=1046.216,48.283,418.520,170.243,35.190,156.623
C04993=1046.223,48.531,418.503,170.244,35.192,156.623
C04994=1046.229,48.781,418.485,170.246,35.193,156.624
C04995=1046.235,49.030,418.469,170.248,35.194,156.624
C04996=1046.242,49.280,418.452,170.249,35.196,156.624
C04997=1046.247,49.529,418.434,170.251,35.198,156.624
C04998=1046.254,49.779,418.418,170.254,35.200,156.625
C04999=1046.260,50.028,418.401,170.255,35.201,156.625
C05000=1046.266,50.277,418.383,170.257,35.203,156.625
C05001=1046.272,50.526,418.366,170.259,35.204,156.625
C05002=1046.279,50.776,418.349,170.260,35.206,156.626
C05003=1046.284,51.025,418.332,170.262,35.207,156.626
C05004=1046.291,51.275,418.314,170.264,35.209,156.626
C05005=1046.297,51.524,418.297,170.265,35.211,156.627
C05006=1046.303,51.774,418.280,170.267,35.212,156.627
C05007=1046.309,52.022,418.263,170.270,35.214,156.627
C05008=1046.316,52.272,418.245,170.271,35.215,156.627
C05009=1046.322,52.521,418.228,170.273,35.217,156.628
C05010=1046.329,52.770,418.211,170.275,35.218,156.628
C05011=1046.334,53.020,418.194,170.276,35.220,156.628
C05012=1046.341,53.269,418.177,170.278,35.222,156.628
C05013=1046.347,53.518,418.160,170.280,35.223,156.629
C05014=1046.353,53.768,418.142,170.281,35.225,156.629
C05015=1046.359,54.017,418.125,170.283,35.226,156.629
C05016=1046.365,54.267,418.108,170.284,35.227,156.629
C05017=1046.371,54.516,418.091,170.287,35.229,156.630
C05018=1046.378,54.765,418.073,170.289,35.231,156.630
C05019=1046.384,55.014,418.056,170.290,35.233,156.630
C05020=1046.391,55.264,418.038,170.292,35.234,156.631
C05021=1046.397,55.513,418.020,170.294,35.236,156.631
C05022=1046.403,55.762,418.003,170.295,35.237,156.631
C05023=1046.410,56.012,417.986,170.297,35.238,156.631
C05024=1046.415,56.261,417.969,170.299,35.240,156.632
C05025=1046.422,56.511,417.952,170.300,35.242,156.632
C05026=1046.428,56.759,417.935,170.302,35.244,156.632
C05027=1046.434,57.009,417.917,170.305,35.245,156.632
C05028=1046.441,57.259,417.900,170.306,35.246,156.633
C05029=1046.447,57.508,417.882,170.308,35.248,156.633
C05030=1046.454,57.757,417.865,170.310,35.249,156.633
C05031=1046.460,58.006,417.848,170.311,35.251,156.633
C05032=1046.466,58.255,417.830,170.313,35.253,156.634
C05033=1046.473,58.505,417.813,170.315,35.254,156.634
C05034=1046.478,58.754,417.795,170.316,35.256,156.634
C05035=1046.485,59.003,417.778,170.318,35.257,156.635
C05036=1046.491,59.253,417.760,170.320,35.259,156.635
C05037=1046.498,59.502,417.743,170.322,35.260,156.635
C05038=1046.504,59.751,417.725,170.324,35.262,156.635
C05039=1046.511,60.001,417.707,170.326,35.264,156.636
C05040=1046.517,60.250,417.691,170.327,35.265,156.636
C05041=1046.523,60.500,417.673,170.329,35.266,156.636
C05042=1046.530,60.749,417.655,170.331,35.268,156.636
C05043=1046.537,61.035,417.635,170.333,35.270,156.637
C05044=1046.544,61.321,417.615,170.334,35.271,156.637
C05045=1046.551,61.607,417.595,170.336,35.273,156.637
C05046=1046.559,61.893,417.574,170.339,35.275,156.638
C05047=1046.565,62.142,417.557,170.341,35.277,156.638
C05048=1046.571,62.391,417.539,170.343,35.278,156.638
C05049=1046.578,62.641,417.522,170.344,35.280,156.638
C05050=1046.585,62.890,417.505,170.346,35.281,156.639
C05051=1046.591,63.140,417.487,170.348,35.282,156.639
C05052=1046.597,63.389,417.470,170.349,35.284,156.639
C05053=1046.603,63.638,417.452,170.351,35.286,156.639
C05054=1046.610,63.888,417.435,170.353,35.287,156.640
C05055=1046.616,64.136,417.416,170.354,35.289,156.640
C05056=1046.623,64.386,417.399,170.357,35.290,156.640
C05057=1046.629,64.635,417.381,170.359,35.292,156.641
C05058=1046.635,64.885,417.363,170.360,35.293,156.641
C05059=1046.641,65.134,417.346,170.362,35.295,156.641
C05060=1046.648,65.383,417.327,170.363,35.297,156.641
C05061=1046.654,65.633,417.310,170.365,35.299,156.642
C05062=1046.659,65.882,417.292,170.367,35.300,156.642
C05063=1046.666,66.131,417.275,170.368,35.302,156.642
C05064=1046.673,66.380,417.256,170.370,35.303,156.642
C05065=1046.678,66.629,417.238,170.373,35.305,156.643
C05066=1046.685,66.879,417.221,170.374,35.306,156.643
C05067=1046.691,67.128,417.203,170.376,35.308,156.643
C05068=1046.698,67.378,417.185,170.378,35.309,156.644
C05069=1046.703,67.627,417.167,170.379,35.311,156.644
C05070=1046.710,67.876,417.150,170.381,35.313,156.644
C05071=1046.716,68.125,417.131,170.382,35.315,156.644
C05072=1046.722,68.375,417.113,170.384,35.316,156.645
C05073=1046.728,68.624,417.095,170.386,35.318,156.645
C05074=1046.735,68.873,417.077,170.388,35.319,156.645
C05075=1046.741,69.123,417.059,170.390,35.321,156.646
C05076=1046.747,69.372,417.042,170.392,35.322,156.646
C05077=1046.753,69.621,417.023,170.393,35.324,156.646
C05078=1046.759,69.870,417.005,170.395,35.326,156.646
C05079=1046.765,70.120,416.987,170.397,35.327,156.647
C05080=1046.772,70.368,416.970,170.398,35.329,156.647
C05081=1046.778,70.618,416.952,170.400,35.331,156.647
C05082=1046.785,70.867,416.933,170.402,35.333,156.648
C05083=1046.791,71.117,416.915,170.404,35.334,156.648
C05084=1046.796,71.365,416.897,170.406,35.336,156.648
C05085=1046.803,71.615,416.879,170.407,35.337,156.648
C05086=1046.809,71.865,416.861,170.409,35.339,156.649
C05087=1046.815,72.114,416.842,170.411,35.340,156.649
C05088=1046.821,72.364,416.824,170.412,35.342,156.649
C05089=1046.827,72.612,416.806,170.414,35.343,156.650
C05090=1046.834,72.861,416.789,170.416,35.345,156.650
C05091=1046.840,73.111,416.770,170.418,35.347,156.650
C05092=1046.846,73.360,416.752,170.420,35.349,156.650
C05093=1046.852,73.609,416.734,170.421,35.351,156.651
C05094=1046.858,73.859,416.716,170.423,35.352,156.651
C05095=1046.865,74.108,416.697,170.425,35.354,156.651
C05096=1046.871,74.357,416.679,170.426,35.355,156.652
C05097=1046.877,74.606,416.661,170.428,35.357,156.652
C05098=1046.883,74.856,416.643,170.430,35.358,156.652
C05099=1046.889,75.105,416.625,170.431,35.360,156.652
C05100=1046.896,75.354,416.606,170.434,35.361,156.653
C05101=1046.902,75.604,416.588,170.436,35.363,156.653
C05102=1046.908,75.853,416.569,170.437,35.365,156.653
C05103=1046.914,76.102,416.551,170.439,35.367,156.654
C05104=1046.920,76.351,416.533,170.440,35.368,156.654
C05105=1046.927,76.600,416.516,170.442,35.370,156.654
C05106=1046.934,76.849,416.497,170.444,35.372,156.654
C05107=1046.941,77.136,416.476,170.446,35.374,156.655
C05108=1046.948,77.421,416.455,170.448,35.375,156.655
C05109=1046.955,77.707,416.433,170.450,35.377,156.655
C05110=1046.961,77.994,416.413,170.452,35.379,156.656
C05111=1046.968,78.243,416.394,170.454,35.381,156.656
C05112=1046.974,78.492,416.375,170.455,35.383,156.656
C05113=1046.980,78.742,416.357,170.457,35.384,156.657
C05114=1046.986,78.990,416.339,170.459,35.386,156.657
C05115=1046.993,79.239,416.321,170.460,35.387,156.657
C05116=1046.999,79.488,416.302,170.463,35.389,156.658
C05117=1047.004,79.738,416.283,170.465,35.391,156.658
C05118=1047.011,79.987,416.265,170.466,35.392,156.658
C05119=1047.017,80.236,416.246,170.468,35.394,156.658
C05120=1047.024,80.486,416.227,170.469,35.396,156.659
C05121=1047.029,80.735,416.210,170.471,35.397,156.659
C05122=1047.036,80.984,416.191,170.473,35.399,156.659
C05123=1047.041,81.233,416.172,170.474,35.401,156.660
C05124=1047.048,81.482,416.153,170.477,35.402,156.660
C05125=1047.054,81.732,416.135,170.479,35.404,156.660
C05126=1047.060,81.981,416.117,170.480,35.406,156.660
C05127=1047.067,82.230,416.098,170.482,35.407,156.661
C05128=1047.072,82.480,416.079,170.483,35.409,156.661
C05129=1047.079,82.729,416.060,170.485,35.411,156.661
C05130=1047.084,82.978,416.043,170.487,35.413,156.662
C05131=1047.091,83.227,416.024,170.488,35.414,156.662
C05132=1047.096,83.476,416.005,170.490,35.416,156.662
C05133=1047.103,83.726,415.986,170.493,35.418,156.663
C05134=1047.109,83.975,415.967,170.494,35.419,156.663
C05135=1047.116,84.224,415.949,170.496,35.421,156.663
C05136=1047.122,84.473,415.930,170.498,35.423,156.664
C05137=1047.127,84.723,415.912,170.499,35.424,156.664
C05138=1047.134,84.972,415.893,170.501,35.426,156.664
C05139=1047.140,85.221,415.874,170.502,35.427,156.664
C05140=1047.147,85.470,415.856,170.504,35.429,156.665
C05141=1047.152,85.720,415.836,170.507,35.431,156.665
C05142=1047.159,85.969,415.818,170.508,35.432,156.665
C05143=1047.165,86.218,415.799,170.510,35.434,156.666
C05144=1047.172,86.467,415.780,170.512,35.436,156.666
C05145=1047.177,86.717,415.761,170.513,35.437,156.666
C05146=1047.184,86.966,415.743,170.515,35.439,156.666
C05147=1047.190,87.215,415.724,170.517,35.441,156.667
C05148=1047.197,87.464,415.705,170.518,35.443,156.667
C05149=1047.202,87.713,415.686,170.521,35.444,156.667
C05150=1047.209,87.963,415.667,170.523,35.446,156.668
C05151=1047.215,88.212,415.649,170.524,35.447,156.668
C05152=1047.222,88.461,415.630,170.526,35.449,156.668
C05153=1047.227,88.710,415.611,170.527,35.451,156.669
C05154=1047.234,88.959,415.592,170.529,35.452,156.669
C05155=1047.240,89.208,415.574,170.531,35.454,156.669
C05156=1047.247,89.458,415.555,170.532,35.455,156.669
C05157=1047.252,89.707,415.536,170.535,35.457,156.670
C05158=1047.259,89.956,415.517,170.537,35.459,156.670
C05159=1047.265,90.205,415.498,170.538,35.460,156.670
C05160=1047.272,90.454,415.480,170.540,35.462,156.671
C05161=1047.277,90.704,415.460,170.542,35.464,156.671
C05162=1047.284,90.953,415.442,170.543,35.466,156.671
C05163=1047.289,91.202,415.423,170.545,35.467,156.671
C05164=1047.296,91.451,415.404,170.548,35.469,156.672
C05165=1047.302,91.701,415.385,170.549,35.471,156.672
C05166=1047.308,91.950,415.365,170.551,35.473,156.672
C05167=1047.314,92.199,415.346,170.552,35.474,156.673
C05168=1047.320,92.448,415.327,170.554,35.476,156.673
C05169=1047.326,92.697,415.308,170.556,35.478,156.673
C05170=1047.332,92.947,415.289,170.557,35.480,156.674
C05171=1047.339,93.233,415.267,170.559,35.481,156.674
C05172=1047.346,93.518,415.245,170.562,35.483,156.674
C05173=1047.353,93.804,415.223,170.564,35.485,156.675
C05174=1047.360,94.090,415.201,170.566,35.487,156.675
C05175=1047.366,94.340,415.182,170.568,35.489,156.675
C05176=1047.373,94.588,415.163,170.569,35.490,156.676
C05177=1047.378,94.838,415.144,170.571,35.492,156.676
C05178=1047.385,95.087,415.125,170.572,35.494,156.676
C05179=1047.391,95.336,415.106,170.575,35.495,156.677
C05180=1047.397,95.585,415.086,170.577,35.497,156.677
C05181=1047.403,95.834,415.067,170.578,35.499,156.677
C05182=1047.409,96.083,415.048,170.580,35.500,156.677
C05183=1047.415,96.333,415.029,170.582,35.502,156.678
C05184=1047.422,96.582,415.009,170.583,35.504,156.678
C05185=1047.428,96.831,414.990,170.585,35.506,156.678
C05186=1047.434,97.080,414.972,170.587,35.507,156.679
C05187=1047.440,97.329,414.952,170.589,35.509,156.679
C05188=1047.446,97.579,414.932,170.591,35.511,156.679
C05189=1047.453,97.828,414.914,170.593,35.513,156.680
C05190=1047.459,98.077,414.894,170.594,35.514,156.680
C05191=1047.465,98.326,414.875,170.596,35.516,156.680
C05192=1047.471,98.576,414.855,170.598,35.518,156.681
C05193=1047.478,98.824,414.836,170.599,35.520,156.681
C05194=1047.484,99.074,414.817,170.601,35.521,156.681
C05195=1047.489,99.323,414.798,170.604,35.523,156.681
C05196=1047.496,99.572,414.778,170.605,35.525,156.682
C05197=1047.502,99.821,414.759,170.607,35.526,156.682
C05198=1047.508,100.070,414.740,170.609,35.528,156.682
C05199=1047.515,100.320,414.720,170.610,35.530,156.683
C05200=1047.521,100.569,414.701,170.612,35.531,156.683
C05201=1047.527,100.818,414.681,170.614,35.533,156.683
C05202=1047.533,101.067,414.662,170.616,35.535,156.684
C05203=1047.539,101.316,414.642,170.618,35.537,156.684
C05204=1047.545,101.565,414.623,170.619,35.538,156.684
C05205=1047.552,101.815,414.603,170.621,35.540,156.685
C05206=1047.558,102.064,414.584,170.623,35.542,156.685
C05207=1047.564,102.313,414.564,170.624,35.544,156.685
C05208=1047.569,102.562,414.545,170.626,35.545,156.685
C05209=1047.575,102.811,414.525,170.629,35.547,156.686
C05210=1047.582,103.060,414.506,170.630,35.549,156.686
C05211=1047.588,103.309,414.486,170.632,35.551,156.686
C05212=1047.594,103.559,414.467,170.634,35.552,156.687
C05213=1047.600,103.808,414.447,170.635,35.554,156.687
C05214=1047.606,104.057,414.427,170.637,35.556,156.687
C05215=1047.612,104.306,414.407,170.639,35.558,156.688
C05216=1047.618,104.555,414.388,170.641,35.559,156.688
C05217=1047.625,104.805,414.368,170.643,35.561,156.688
C05218=1047.631,105.054,414.349,170.645,35.563,156.689
C05219=1047.636,105.303,414.329,170.646,35.565,156.689
C05220=1047.642,105.552,414.309,170.648,35.566,156.689
C05221=1047.648,105.801,414.289,170.650,35.568,156.690
C05222=1047.655,106.050,414.270,170.651,35.570,156.690
C05223=1047.661,106.299,414.250,170.654,35.571,156.690
C05224=1047.667,106.549,414.231,170.656,35.573,156.690
C05225=1047.673,106.798,414.211,170.657,35.575,156.691
C05226=1047.679,107.046,414.191,170.659,35.577,156.691
C05227=1047.685,107.297,414.172,170.661,35.578,156.692
C05228=1047.692,107.545,414.152,170.662,35.580,156.692
C05229=1047.698,107.794,414.132,170.664,35.582,156.692
C05230=1047.704,108.043,414.113,170.666,35.584,156.692
C05231=1047.710,108.293,414.093,170.668,35.585,156.693
C05232=1047.716,108.542,414.073,170.670,35.587,156.693
C05233=1047.722,108.790,414.053,170.672,35.589,156.693
C05234=1047.729,109.041,414.033,170.673,35.590,156.694
C05235=1047.736,109.326,414.011,170.675,35.592,156.694
C05236=1047.743,109.612,413.988,170.677,35.594,156.694
C05237=1047.751,109.897,413.965,170.680,35.596,156.695
C05238=1047.757,110.183,413.942,170.682,35.598,156.695
C05239=1047.764,110.432,413.923,170.684,35.600,156.695
C05240=1047.770,110.681,413.903,170.686,35.601,156.696
C05241=1047.776,110.931,413.883,170.687,35.603,156.696
C05242=1047.782,111.180,413.863,170.689,35.605,156.696
C05243=1047.788,111.428,413.843,170.691,35.607,156.697
C05244=1047.794,111.678,413.824,170.693,35.609,156.697
C05245=1047.801,111.927,413.803,170.695,35.610,156.697
C05246=1047.807,112.176,413.784,170.697,35.612,156.698
C05247=1047.813,112.425,413.764,170.698,35.614,156.698
C05248=1047.819,112.675,413.743,170.700,35.616,156.698
C05249=1047.825,112.923,413.723,170.702,35.617,156.699
C05250=1047.831,113.173,413.704,170.703,35.619,156.699
C05251=1047.837,113.422,413.684,170.706,35.621,156.699
C05252=1047.843,113.671,413.664,170.708,35.623,156.700
C05253=1047.849,113.920,413.643,170.709,35.625,156.700
C05254=1047.855,114.170,413.623,170.711,35.626,156.700
C05255=1047.861,114.419,413.603,170.713,35.628,156.701
C05256=1047.867,114.667,413.583,170.714,35.630,156.701
C05257=1047.873,114.916,413.562,170.716,35.632,156.701
C05258=1047.879,115.166,413.542,170.719,35.633,156.702
C05259=1047.885,115.415,413.522,170.720,35.635,156.702
C05260=1047.890,115.664,413.502,170.722,35.637,156.702
C05261=1047.897,115.913,413.481,170.724,35.639,156.703
C05262=1047.903,116.162,413.461,170.725,35.641,156.703
C05263=1047.909,116.411,413.441,170.727,35.643,156.703
C05264=1047.915,116.661,413.420,170.729,35.644,156.704
C05265=1047.921,116.910,413.400,170.731,35.646,156.704
C05266=1047.927,117.159,413.380,170.733,35.648,156.704
C05267=1047.933,117.408,413.360,170.735,35.650,156.705
C05268=1047.939,117.657,413.340,170.737,35.652,156.705
C05269=1047.945,117.906,413.320,170.738,35.654,156.705
C05270=1047.951,118.155,413.299,170.740,35.655,156.706
C05271=1047.956,118.405,413.279,170.743,35.657,156.706
C05272=1047.963,118.653,413.258,170.744,35.659,156.706
C05273=1047.969,118.902,413.238,170.746,35.660,156.707
C05274=1047.975,119.151,413.218,170.748,35.662,156.707
C05275=1047.981,119.400,413.197,170.749,35.664,156.707
C05276=1047.987,119.650,413.177,170.751,35.666,156.708
C05277=1047.993,119.899,413.157,170.754,35.668,156.708
C05278=1047.999,120.148,413.136,170.755,35.670,156.708
C05279=1048.005,120.397,413.116,170.757,35.672,156.709
C05280=1048.011,120.645,413.095,170.759,35.674,156.709
C05281=1048.017,120.895,413.074,170.761,35.675,156.709
C05282=1048.023,121.144,413.055,170.762,35.677,156.710
C05283=1048.030,121.394,413.034,170.764,35.679,156.710
C05284=1048.035,121.643,413.014,170.767,35.681,156.710
C05285=1048.041,121.891,412.993,170.768,35.682,156.711
C05286=1048.048,122.140,412.973,170.770,35.684,156.711
C05287=1048.054,122.389,412.953,170.772,35.686,156.711
C05288=1048.060,122.639,412.932,170.774,35.688,156.712
C05289=1048.066,122.888,412.912,170.775,35.689,156.712
C05290=1048.073,123.137,412.891,170.777,35.691,156.712
C05291=1048.078,123.386,412.870,170.780,35.693,156.713
C05292=1048.085,123.635,412.850,170.781,35.695,156.713
C05293=1048.091,123.884,412.830,170.783,35.697,156.713
C05294=1048.097,124.133,412.808,170.785,35.699,156.714
C05295=1048.103,124.382,412.788,170.787,35.700,156.714
C05296=1048.109,124.631,412.768,170.788,35.702,156.714
C05297=1048.115,124.880,412.747,170.791,35.704,156.715
C05298=1048.121,125.129,412.727,170.793,35.706,156.715
C05299=1048.128,125.415,412.703,170.795,35.708,156.715
C05300=1048.135,125.701,412.680,170.797,35.710,156.716
C05301=1048.142,125.987,412.656,170.799,35.712,156.716
C05302=1048.149,126.272,412.633,170.801,35.714,156.716
C05303=1048.155,126.522,412.612,170.804,35.716,156.717
C05304=1048.161,126.770,412.591,170.805,35.718,156.717
C05305=1048.168,127.019,412.571,170.807,35.719,156.717
C05306=1048.174,127.269,412.550,170.809,35.721,156.718
C05307=1048.180,127.517,412.529,170.811,35.723,156.718
C05308=1048.187,127.767,412.509,170.812,35.725,156.718
C05309=1048.192,128.016,412.487,170.815,35.726,156.719
C05310=1048.199,128.265,412.467,170.817,35.728,156.719
C05311=1048.204,128.514,412.447,170.819,35.730,156.719
C05312=1048.211,128.763,412.425,170.820,35.732,156.720
C05313=1048.217,129.012,412.406,170.822,35.733,156.720
C05314=1048.223,129.261,412.384,170.824,35.735,156.720
C05315=1048.230,129.511,412.364,170.826,35.737,156.721
C05316=1048.236,129.759,412.343,170.828,35.738,156.721
C05317=1048.242,130.009,412.322,170.830,35.740,156.721
C05318=1048.248,130.257,412.302,170.832,35.742,156.722
C05319=1048.254,130.507,412.280,170.834,35.744,156.722
C05320=1048.261,130.756,412.260,170.835,35.746,156.722
C05321=1048.267,131.004,412.239,170.837,35.748,156.723
C05322=1048.273,131.254,412.218,170.840,35.749,156.723
C05323=1048.279,131.502,412.198,170.842,35.751,156.723
C05324=1048.285,131.752,412.176,170.843,35.753,156.724
C05325=1048.291,132.001,412.155,170.845,35.755,156.724
C05326=1048.297,132.250,412.135,170.847,35.757,156.724
C05327=1048.303,132.499,412.114,170.849,35.758,156.725
C05328=1048.309,132.748,412.092,170.852,35.760,156.725
C05329=1048.315,132.997,412.072,170.853,35.762,156.725
C05330=1048.321,133.246,412.051,170.855,35.764,156.726
C05331=1048.327,133.495,412.029,170.857,35.766,156.726
C05332=1048.334,133.745,412.009,170.859,35.768,156.726
C05333=1048.339,133.993,411.988,170.860,35.770,156.727
C05334=1048.345,134.242,411.966,170.863,35.772,156.727
C05335=1048.351,134.491,411.946,170.865,35.774,156.727
C05336=1048.358,134.740,411.924,170.867,35.775,156.728
C05337=1048.364,134.990,411.903,170.868,35.777,156.728
C05338=1048.370,135.238,411.883,170.870,35.779,156.729
C05339=1048.376,135.488,411.861,170.872,35.781,156.729
C05340=1048.382,135.737,411.839,170.875,35.783,156.729
C05341=1048.388,135.986,411.819,170.876,35.785,156.730
C05342=1048.394,136.235,411.798,170.878,35.786,156.730
C05343=1048.400,136.483,411.777,170.880,35.788,156.730
C05344=1048.407,136.732,411.756,170.882,35.790,156.731
C05345=1048.413,136.982,411.735,170.884,35.792,156.731
C05346=1048.418,137.231,411.713,170.885,35.794,156.731
C05347=1048.424,137.480,411.692,170.888,35.795,156.732
C05348=1048.431,137.729,411.671,170.890,35.797,156.732
C05349=1048.437,137.977,411.649,170.892,35.799,156.732
C05350=1048.443,138.227,411.628,170.894,35.801,156.733
C05351=1048.449,138.476,411.607,170.895,35.803,156.733
C05352=1048.455,138.724,411.586,170.898,35.805,156.733
C05353=1048.461,138.974,411.565,170.900,35.807,156.734
C05354=1048.467,139.223,411.543,170.902,35.809,156.734
C05355=1048.473,139.472,411.522,170.904,35.810,156.734
C05356=1048.479,139.721,411.501,170.905,35.812,156.735
C05357=1048.486,139.970,411.480,170.907,35.814,156.735
C05358=1048.492,140.219,411.458,170.910,35.816,156.735
C05359=1048.497,140.468,411.437,170.912,35.818,156.736
C05360=1048.504,140.717,411.415,170.913,35.820,156.736
C05361=1048.510,140.966,411.394,170.915,35.822,156.737
C05362=1048.515,141.215,411.372,170.917,35.824,156.737
C05363=1048.522,141.501,411.348,170.919,35.826,156.737
C05364=1048.530,141.786,411.323,170.922,35.828,156.738
C05365=1048.536,142.072,411.299,170.924,35.830,156.738
C05366=1048.543,142.357,411.274,170.926,35.832,156.739
C05367=1048.549,142.606,411.252,170.928,35.834,156.739
C05368=1048.555,142.855,411.231,170.930,35.836,156.739
C05369=1048.561,143.104,411.209,170.933,35.838,156.740
C05370=1048.568,143.353,411.188,170.935,35.840,156.740
C05371=1048.573,143.602,411.167,170.936,35.842,156.740
C05372=1048.580,143.851,411.145,170.938,35.844,156.741
C05373=1048.586,144.100,411.124,170.940,35.846,156.741
C05374=1048.592,144.349,411.102,170.942,35.848,156.741
C05375=1048.597,144.598,411.081,170.945,35.850,156.742
C05376=1048.604,144.847,411.059,170.946,35.852,156.742
C05377=1048.610,145.096,411.037,170.948,35.853,156.743
C05378=1048.616,145.345,411.016,170.950,35.855,156.743
C05379=1048.622,145.595,410.994,170.952,35.857,156.743
C05380=1048.628,145.843,410.973,170.954,35.859,156.744
C05381=1048.634,146.092,410.950,170.957,35.861,156.744
C05382=1048.640,146.341,410.929,170.958,35.863,156.744
C05383=1048.646,146.590,410.907,170.960,35.865,156.745
C05384=1048.653,146.839,410.886,170.962,35.867,156.745
C05385=1048.658,147.088,410.864,170.964,35.868,156.745
C05386=1048.664,147.337,410.843,170.967,35.870,156.746
C05387=1048.670,147.586,410.821,170.969,35.872,156.746
C05388=1048.677,147.835,410.799,170.971,35.874,156.746
C05389=1048.683,148.084,410.777,170.972,35.876,156.747
C05390=1048.689,148.332,410.756,170.974,35.878,156.747
C05391=1048.695,148.582,410.734,170.976,35.880,156.748
C05392=1048.701,148.831,410.713,170.979,35.882,156.748
C05393=1048.707,149.080,410.690,170.981,35.884,156.748
C05394=1048.713,149.329,410.668,170.983,35.886,156.749
C05395=1048.718,149.577,410.647,170.984,35.888,156.749
C05396=1048.725,149.827,410.625,170.986,35.890,156.749
C05397=1048.731,150.075,410.603,170.989,35.891,156.750
C05398=1048.737,150.324,410.581,170.991,35.894,156.750
C05399=1048.743,150.574,410.559,170.993,35.896,156.751
C05400=1048.749,150.823,410.536,170.995,35.898,156.751
C05401=1048.755,151.071,410.515,170.997,35.900,156.751
C05402=1048.761,151.320,410.494,170.998,35.901,156.752
C05403=1048.767,151.569,410.471,171.001,35.903,156.752
C05404=1048.773,151.818,410.449,171.003,35.905,156.752
C05405=1048.779,152.068,410.427,171.005,35.908,156.753
C05406=1048.785,152.316,410.405,171.007,35.909,156.753
C05407=1048.792,152.565,410.383,171.009,35.911,156.753
C05408=1048.796,152.814,410.361,171.012,35.913,156.754
C05409=1048.803,153.063,410.339,171.013,35.915,156.754
C05410=1048.809,153.312,410.317,171.015,35.917,156.755
C05411=1048.815,153.561,410.296,171.017,35.919,156.755
C05412=1048.822,153.810,410.274,171.019,35.921,156.755
C05413=1048.827,154.059,410.251,171.022,35.923,156.756
C05414=1048.834,154.308,410.229,171.024,35.925,156.756
C05415=1048.840,154.557,410.207,171.026,35.927,156.756
C05416=1048.846,154.806,410.185,171.028,35.929,156.757
C05417=1048.852,155.055,410.163,171.029,35.931,156.757
C05418=1048.858,155.304,410.140,171.032,35.933,156.758
C05419=1048.863,155.553,410.118,171.034,35.935,156.758
C05420=1048.869,155.801,410.096,171.036,35.937,156.758
C05421=1048.876,156.050,410.075,171.038,35.939,156.759
C05422=1048.881,156.299,410.052,171.040,35.941,156.759
C05423=1048.887,156.549,410.030,171.042,35.943,156.760
C05424=1048.894,156.797,410.008,171.045,35.945,156.760
C05425=1048.899,157.047,409.985,171.047,35.947,156.760
C05426=1048.906,157.295,409.963,171.048,35.949,156.761
C05427=1048.912,157.580,409.938,171.051,35.951,156.761
C05428=1048.920,157.865,409.912,171.053,35.954,156.762
C05429=1048.926,158.151,409.887,171.056,35.955,156.762
C05430=1048.934,158.436,409.862,171.058,35.958,156.762
C05431=1048.939,158.685,409.839,171.060,35.960,156.763
C05432=1048.946,158.934,409.816,171.062,35.962,156.763
C05433=1048.951,159.183,409.794,171.065,35.964,156.764
C05434=1048.958,159.432,409.772,171.067,35.966,156.764
C05435=1048.964,159.680,409.749,171.069,35.968,156.764
C05436=1048.970,159.930,409.727,171.071,35.970,156.765
C05437=1048.976,160.179,409.705,171.073,35.972,156.765
C05438=1048.982,160.427,409.682,171.075,35.974,156.765
C05439=1048.988,160.677,409.660,171.077,35.976,156.766
C05440=1048.994,160.926,409.637,171.079,35.978,156.766
C05441=1048.999,161.174,409.614,171.081,35.980,156.767
C05442=1049.006,161.423,409.592,171.083,35.982,156.767
C05443=1049.011,161.673,409.570,171.086,35.985,156.767
C05444=1049.017,161.921,409.547,171.088,35.986,156.768
C05445=1049.023,162.170,409.524,171.090,35.988,156.768
C05446=1049.028,162.419,409.501,171.092,35.991,156.769
C05447=1049.035,162.668,409.479,171.094,35.993,156.769
C05448=1049.040,162.917,409.457,171.097,35.995,156.769
C05449=1049.045,163.166,409.434,171.098,35.997,156.770
C05450=1049.051,163.414,409.411,171.100,35.999,156.770
C05451=1049.058,163.663,409.389,171.102,36.001,156.771
C05452=1049.063,163.912,409.366,171.104,36.003,156.771
C05453=1049.069,164.161,409.343,171.107,36.006,156.772
C05454=1049.075,164.410,409.320,171.109,36.007,156.772
C05455=1049.081,164.659,409.297,171.111,36.010,156.772
C05456=1049.087,164.908,409.275,171.113,36.012,156.773
C05457=1049.093,165.157,409.252,171.115,36.014,156.773
C05458=1049.098,165.406,409.229,171.118,36.016,156.774
C05459=1049.104,165.655,409.206,171.120,36.018,156.774
C05460=1049.110,165.903,409.184,171.122,36.020,156.774
C05461=1049.117,166.153,409.161,171.124,36.022,156.775
C05462=1049.122,166.402,409.138,171.127,36.025,156.775
C05463=1049.128,166.651,409.115,171.128,36.027,156.776
C05464=1049.134,166.899,409.092,171.130,36.028,156.776
C05465=1049.140,167.148,409.069,171.132,36.031,156.776
C05466=1049.146,167.397,409.046,171.134,36.033,156.777
